//Roby - Alterado em 29/08/2020==========================INICIO==========================
// Entrada analógica 01 : NX6000_3 - %IW80 - Medição da temperatura da ENTRADA DA TORRE com SENSOR TIPO K e TXBLOCK =========================== 
converteEA103(IN:=EA103, IN_MIN:=0, IN_MAX:=4000,OUT_MIN:= -150, OUT_MAX:=1370);
TEMP_QUEIMATORRE:= converteEA103.OUT;

// Entrada analógica 02 : NX6000_3 - %IW82 - Medição da temperatura da SAÍDA ATMOSFERA com SENSOR TIPO K e TXBLOCK =========================== 
converteEA203(IN:=EA203, IN_MIN:=0, IN_MAX:=4000,OUT_MIN:= -150, OUT_MAX:=1370);
TEMP_QUEIMAATM:= converteEA203.OUT;

//Roby - Alterado em 23/02/2021==========================INÍCO==========================

// Entrada analógica 03 : NX6000_3 - %IW86 - Transdutor de pressão da tubulação óleo BPF. =========================== 
converteEA403(IN:=EA403, IN_MIN:=0, IN_MAX:=4000,OUT_MIN:=0, OUT_MAX:=16);
PRESS_OLEO_BPF:= converteEA403.OUT;
//Roby - Alterado em 23/02/2021==========================FIM==========================

// Entrada analógica 4 : NX6000_2 - Leitura Fluxo BBP02 ( dm³/h mA) ======================================================= 
converteEA502(IN:=EA502, IN_MIN:=0, IN_MAX:=4000,OUT_MIN:=0, OUT_MAX:=120);
VAZAO_VOLUMETRICA_REAL_BBP02:= converteEA502.OUT;

// Entrada analógica 4 : NX6000_2 - Leitura Fluxo BBP01 ( dm³/h mA) ======================================================= 
converteEA702(IN:=EA702, IN_MIN:=0, IN_MAX:=4000,OUT_MIN:=0, OUT_MAX:=120);
VAZAO_VOLUMETRICA_REAL_BBP01:= converteEA702.OUT;

END_PROGRAM

// Device/Application/BBP02
PROGRAM BBP02
VAR
	// Vazão volumetrica BBP02
	VAZAO_VOLUMETRICA_PRESET: REAL;
	// Vazão massica BBP02 kg/h
	VAZAO_MASSICA: REAL;
	//massa de dosagem do equipamento em Tonelada.
	MASSA:REAL;
	//Velocidade calculda do Dosador em Hz
	VELOCIDADE:REAL;
	//Espera o fluidizador baixar para o peso minino, pois atingiu o peso maximo
	ESPERA_FLUIDIZADOR_BAIXAR_PESO:BOOL;
	//Liga Dosador manual
	LIGA_DS_MANUAL:BOOL;
	//Liga Dosador automatico
	LIGA_DS_AUTO:BOOL;
	//Função de pulso do perfume
	PULSO_PERFUME:R_TRIG;
	// PID da BBP02
	PID_BBP02: NextoPID.PID;
	// constante
	A: BOOL;
	TMR_ATRASO_PERFUME: TON;
	INICIA_ATRASO_PERFUME: BOOL;
END_VAR

//   POU da bomba de perfume 2

//Controle manual ==========================================================

IF BTS_MAPH2 = FALSE THEN		
	
	//Bomba de perfume ===============================================
	//Formula
	//    Passo 1:     massa := (tonelada de dosagem * Percentual de dosagem(sem conversao)  * 10)  
	//    Passo 2:    Velocidade := ((massa + PRST_CONSTANTE_A_BBP02)/PRST_CONSTANTE_B_BBP02 
	//	  Inicialmente a Constante a:= -1.5
	//	  Inicialmente a Constante b:= 2.2948    	

	//calculo de velocidade  ======================================================
	IF MASSA_ESPECIFICA_BBP02 = 0 THEN
	MASSA_ESPECIFICA_BBP02 := 1;
	END_IF
	//Calcuulo da massa de dosagem do equipamento 
	MASSA := (PRST_VEL_PH2_MANUAL * 10 * PRST_PERC_DOSA_BBP02)/ MASSA_ESPECIFICA_BBP02;
	VAZAO_MASSICA := MASSA * MASSA_ESPECIFICA_BBP02;
	//Calculo da velocidade
	//VELOCIDADE := (MASSA + PRST_CONSTANTE_A_BBP02)/PRST_CONSTANTE_B_BBP02; 
	VELOCIDADE := MASSA; 
	IF BTS_BP2 = TRUE  AND AL_GERAL = FALSE   THEN
		IF LIGA_DS_MANUAL = TRUE THEN
			LIGA_DS_MANUAL := FALSE;
		ELSE
			LIGA_DS_MANUAL := TRUE;
		END_IF
		BTS_BP2 := FALSE;
	ELSIF AL_GERAL = TRUE THEN   //delsiga em caso de alarme
		LIGA_DS_MANUAL := FALSE;
		BTS_BP2 := FALSE;
	END_IF		
	
	//velocidde
	PRST_VEL_BPF2 := VELOCIDADE;
	VEL_PROGRAMADA_BBP02 := VAZAO_MASSICA;
	A := FALSE;
		
	//em manual desliga comando do automatico
	LIGA_DS_AUTO := FALSE;
ELSE	
	// controle automatico  =======================================================
		
	//Bomba de perfume ===============================================
	//Formula
	//    Passo 1:     massa := (tonelada de dosagem * Percentual de dosagem(sem conversao)  * 10)  
	//    Passo 2:    Velocidade := ((massa + PRST_CONSTANTE_A_BBP02)/PRST_CONSTANTE_B_BBP02 
	//	  Inicialmente a Constante a:= -1.5
	//	  Inicialmente a Constante b:= 2.2948    	

	//calculo de velocidade  ======================================================

	//Calcuulo da massa de dosagem do equipamento 
	MASSA := ((VELOCIDADE_PH2_AUTO/1000) * 10 * PRST_PERC_DOSA_BBP02)/ MASSA_ESPECIFICA_BBP02 ;
	VAZAO_MASSICA := MASSA;
	
	IF A = FALSE THEN	
		//Calculo da velocidade
		VELOCIDADE := (MASSA + PRST_CONSTANTE_A_BBP02)/PRST_CONSTANTE_B_BBP02; 
		A:=TRUE;
	END_IF	
	
	IF  AL_GERAL = FALSE   THEN		
		LIGA_DS_AUTO := TRUE;
	ELSE
		LIGA_DS_AUTO := FALSE;
	END_IF	
	
	//zera velocidade do ph com peso maximo
	IF LEITURA_PESO_FLUI2 >= PRST_PESO_MAX_FLUID2 THEN
		ESPERA_FLUIDIZADOR_BAIXAR_PESO := TRUE;
	END_IF
	
	//ativa velocidade do ph com peso minimo
	IF LEITURA_PESO_FLUI2 <= PRST_PESO_MIN_FLUID2 THEN
		ESPERA_FLUIDIZADOR_BAIXAR_PESO := FALSE;
	END_IF
	
	//se pode enviar peso 
//se pode enviar peso 
	IF ESPERA_FLUIDIZADOR_BAIXAR_PESO = FALSE THEN
		PRST_VEL_BPF2 := VELOCIDADE;
		VEL_PROGRAMADA_BBP02 := VAZAO_MASSICA;
		IF (VAZAO_VOLUMETRICA_REAL_BBP02 / MASSA_ESPECIFICA_BBP02) < (VAZAO_MASSICA - 1) THEN
			VELOCIDADE := VELOCIDADE + 0.1;
		END_IF
		IF (VAZAO_VOLUMETRICA_REAL_BBP02 / MASSA_ESPECIFICA_BBP02) > (VAZAO_MASSICA + 1) THEN
			VELOCIDADE := VELOCIDADE - 0.1;
		END_IF
		
	ELSE
		PRST_VEL_BPF2 := 0;
		VEL_PROGRAMADA_BBP02 := 0;
	END_IF
	
	//em auto desliga comando do manual
	LIGA_DS_MANUAL := FALSE;	
END_IF

//Liga dosador
IF LIGA_DS_AUTO = TRUE OR LIGA_DS_MANUAL = TRUE THEN
	INICIA_ATRASO_PERFUME := TRUE;
	VEL_BP2 := PRST_VEL_BPF2;
	LEITURA_VEL_BBP2 := VAZAO_VOLUMETRICA_REAL_BBP02/MASSA_ESPECIFICA_BBP02;
ELSE
	INICIA_ATRASO_PERFUME := FALSE;
	SD_BPER2 := FALSE;
	VEL_BP2:= 0;
	LEITURA_VEL_BBP2 := VAZAO_VOLUMETRICA_REAL_BBP02 / MASSA_ESPECIFICA_BBP02;
END_IF

//Atraso na partida da bomba de perfume para esperar chegada do pó.
TMR_ATRASO_PERFUME(IN:=INICIA_ATRASO_PERFUME,PT:= T#60S);
IF 	TMR_ATRASO_PERFUME.Q = TRUE AND LIGA_DS_AUTO = TRUE THEN
SD_BPER2 := TRUE;
END_IF

IF VEL_BP2 = 0 THEN 
	SD_BPER2 := FALSE;
END_IF
 
//Quantidade de consumo do perfume ===========================================

//gera pulso de contagem da agua		
PULSO_PERFUME(CLK:=ED_BP2);

//contador
IF PULSO_PERFUME.Q = TRUE THEN
	
	TOTALIZADOR1_BBP02 := TOTALIZADOR1_BBP02 + (PRST_RAZAO_BPF2 * MASSA_ESPECIFICA_BBP02 * 0.89);
	TOTALIZADOR2_BBP02 := TOTALIZADOR2_BBP02 + (PRST_RAZAO_BPF2 * MASSA_ESPECIFICA_BBP02 * 0.89);
	TOTALIZADOR3_BBP02 := TOTALIZADOR3_BBP02 + (PRST_RAZAO_BPF2 * MASSA_ESPECIFICA_BBP02 * 0.89);
	
END_IF

END_PROGRAM

// Device/Application/PH
PROGRAM PH
VAR
	//Tempos
	
	//Tempo de estrela do exaustor FM1
	TMR_ESTRELA_FM1:TON;
	//Tempo retardo troca de estrela para triangulo exaustor FM1
	TMR_RETARDO_TRIANGULO_FM1:TON;
	//Tempo de estrela do exaustor FM2
	TMR_ESTRELA_FM2:TON;
	//Tempo retardo troca de estrela para triangulo exaustor FM2
	TMR_RETARDO_TRIANGULO_FM2:TON;
	//Tempo de estrela do ventilador FM3
	TMR_ESTRELA_VFM2:TON;
	//Tempo retardo troca de estrela para triangulo ventilador FM2
	TMR_RETARDO_TRIANGULO_VFM2:TON;
	
	//Boleanos
	
	//Libera triangulo exaustor FM1
	LIBERA_TRIANGULO_FM1:BOOL;
	//Liga estrela exaustor FM1
	LIGA_ESTRELA_FM1:BOOL;
	//Liga triangulo exaustor FM1
	LIGA_TRIANGULO_FM1:BOOL;
	//Libera triangulo exaustor FM2
	LIBERA_TRIANGULO_FM2:BOOL;
	//Liga estrela exaustor FM2
	LIGA_ESTRELA_FM2:BOOL;
	//Liga triangulo exaustor FM2
	LIGA_TRIANGULO_FM2:BOOL;
	//Libera triangulo exaustor FM3
	LIBERA_TRIANGULO_VFM2:BOOL;
	//Liga estrela exaustor FM3
	LIGA_ESTRELA_VFM2:BOOL;
	//Liga triangulo exaustor FM3
	LIGA_TRIANGULO_VFM2:BOOL;
	//Liga exaustor FM1
	LIGA_FM1:BOOL;
	//Liga exaustor FM1
	LIGA_FM2:BOOL;
	//Liga ventilador FM2
	LIGA_VENTILADOR_FM2:BOOL;
	//Liga TC13
	LIGA_TC13:BOOL;
END_VAR

//     Processo Powder Handling - lógica do controle do PH

//=================================================================================================
// Controle manual dos equipamentos 
//=================================================================================================

//Controle manual PH 1

IF BTS_MAPH1 = FALSE THEN
	
	// Bomba de alimentação do oelo ===========================================	
	
	IF BTS_BALIOLEO = TRUE  AND AL_GERAL = FALSE  THEN	
		IF SD_BAO = TRUE THEN
			SD_BAO := FALSE;
		ELSE
			SD_BAO := TRUE;	
		END_IF
		 BTS_BALIOLEO := FALSE;
	END_IF
	//desliga em caso de alarme
	IF AL_GERAL = TRUE  THEN
		SD_BAO := FALSE;
		BTS_BALIOLEO := FALSE;
	END_IF
	
ELSE
	//=========================================================================
	// controle automatico PH1 
	//=========================================================================
	
	//Bomba alimentação do óleo ===============================================
	IF AL_GERAL = FALSE AND AL_GERAL = FALSE THEN
		SD_BAO := TRUE;
	ELSE
		SD_BAO := FALSE;
	END_IF
		
END_IF


//=================================================================================================
// Controles que independem do manual/automatico 
//=================================================================================================


// Ventilador do Fluidizador ================================================
//Velocidade  de 0-100%

IF BTS_VENTIFLUIDIZADOR = TRUE  AND AL_GERAL=FALSE THEN
	IF SD_VFLU = TRUE THEN
		SD_VFLU := FALSE;
	ELSE
		SD_VFLU := TRUE;
	END_IF	
	BTS_VENTIFLUIDIZADOR := FALSE;
END_IF
//delsiga em caso de alarme
IF AL_GERAL = TRUE THEN
	SD_VFLU := FALSE;
END_IF

//move velocidade
IF SD_VFLU = TRUE THEN
	VEL_VENTFLUIDIZADOR := PRST_VEL_VENTIFLUIDIZADOR;
ELSE
	VEL_VENTFLUIDIZADOR := 0;
END_IF


//Exaustor FM1 ========================================================

IF BTS_EXFM1 = TRUE AND AL_EXFM1_E = FALSE AND AL_GERAL = FALSE THEN
		IF LIGA_FM1 = TRUE THEN
			LIGA_FM1 := FALSE;
		ELSE
			LIGA_FM1 := TRUE;
		END_IF		
		BTS_EXFM1 := FALSE;	
ELSIF AL_GERAL = TRUE THEN
	LIGA_FM1 := FALSE;
	BTS_EXFM1 := FALSE;
END_IF

//comando estrela/triangulo
//LIGA ESTRELA	
IF LIGA_FM1 = TRUE AND AL_EXFM1_E = FALSE AND  AL_GERAL = FALSE THEN
	IF LIGA_ESTRELA_FM1 = FALSE THEN
		//Contatora estrela
		SD_EXFM1_E := TRUE;
	ELSE
		//Contatora estrela
		SD_EXFM1_E := FALSE;
	END_IF
	LIBERA_TRIANGULO_FM1 := TRUE;
ELSE
	//Contatora estrela
	SD_EXFM1_E := FALSE;	
	LIBERA_TRIANGULO_FM1:=FALSE;
END_IF
	
//TEMPO PARA ENTRAR O TRIANGULO
TMR_ESTRELA_FM1(IN:= LIBERA_TRIANGULO_FM1, PT:= T#6S);	
LIGA_ESTRELA_FM1 := TMR_ESTRELA_FM1.Q;
//TEMPO DE INTERVALO ENTRE ESTRELA E TRIANGULO
TMR_RETARDO_TRIANGULO_FM1(IN:= LIGA_ESTRELA_FM1, PT:= T#0.2S);
LIGA_TRIANGULO_FM1 := TMR_RETARDO_TRIANGULO_FM1.Q;
//Contatora triangulo
SD_EXFM1_T := LIGA_TRIANGULO_FM1;

//contatora Principal	
IF LIBERA_TRIANGULO_FM1 = TRUE THEN
	SD_EXFM1_P := TRUE;
ELSE
	SD_EXFM1_P := FALSE;
END_IF

//Exaustor FM2 ========================================================

IF BTS_EXFM2 = TRUE AND AL_EXFM1_E = FALSE AND AL_GERAL = FALSE THEN
		IF LIGA_FM2 = TRUE THEN
			LIGA_FM2 := FALSE;
		ELSE
			LIGA_FM2 := TRUE;
		END_IF		
		BTS_EXFM2 := FALSE;	
ELSIF AL_GERAL = TRUE THEN
	LIGA_FM2 := FALSE;
	BTS_EXFM2 := FALSE;	
END_IF

//comando estrela/triangulo
//LIGA ESTRELA	
IF LIGA_FM2 = TRUE AND AL_EXFM2_E = FALSE  AND AL_EXFM2_T = FALSE AND AL_GERAL = FALSE THEN
	IF LIGA_ESTRELA_FM2 = FALSE THEN
		//Contatora estrela
		SD_EXFM2_E := TRUE;
	ELSE
		//Contatora estrela
		SD_EXFM2_E := FALSE;
	END_IF
	LIBERA_TRIANGULO_FM2 := TRUE;
ELSE
	//Contatora estrela
	SD_EXFM2_E := FALSE;	
	LIBERA_TRIANGULO_FM2:=FALSE;
END_IF
	
//TEMPO PARA ENTRAR O TRIANGULO
TMR_ESTRELA_FM2(IN:= LIBERA_TRIANGULO_FM2, PT:= T#6S);	
LIGA_ESTRELA_FM2 := TMR_ESTRELA_FM2.Q;
//TEMPO DE INTERVALO ENTRE ESTRELA E TRIANGULO
TMR_RETARDO_TRIANGULO_FM2(IN:= LIGA_ESTRELA_FM2, PT:= T#0.2S);
LIGA_TRIANGULO_FM2 := TMR_RETARDO_TRIANGULO_FM2.Q;
//Contatora triangulo
SD_EXFM2_T := LIGA_TRIANGULO_FM2;

//contatora Principal	
IF LIBERA_TRIANGULO_FM2 = TRUE THEN
	SD_EXFM2_P := TRUE;
ELSE
	SD_EXFM2_P := FALSE;
END_IF


//Ventilador FM1 - PH1 ========================================================

IF BTS_EXVFM2 = TRUE AND AL_EXFM1_E = FALSE AND  AL_GERAL = FALSE THEN
		IF LIGA_VENTILADOR_FM2 = TRUE THEN
			LIGA_VENTILADOR_FM2 := FALSE;
		ELSE
			LIGA_VENTILADOR_FM2 := TRUE;
		END_IF		
		BTS_EXVFM2 := FALSE;
ELSIF  AL_GERAL = TRUE THEN
	LIGA_VENTILADOR_FM2 := FALSE;
	BTS_EXVFM2 := FALSE;
END_IF


//comando estrela/triangulo
//LIGA ESTRELA	
IF LIGA_VENTILADOR_FM2 = TRUE AND AL_VEXFM2_E = FALSE AND AL_VEXFM2_T = FALSE AND  AL_GERAL = FALSE THEN
	IF LIGA_ESTRELA_VFM2 = FALSE THEN
		//Contatora estrela
		SD_VEXFM2_E := TRUE;
	ELSE
		//Contatora estrela
		SD_VEXFM2_E := FALSE;
	END_IF
	LIBERA_TRIANGULO_VFM2 := TRUE;
ELSE
	//Contatora estrela
	SD_VEXFM2_E := FALSE;	
	LIBERA_TRIANGULO_VFM2:=FALSE;
END_IF
	
//TEMPO PARA ENTRAR O TRIANGULO
TMR_ESTRELA_VFM2(IN:= LIBERA_TRIANGULO_VFM2, PT:= T#6S);	
LIGA_ESTRELA_VFM2 := TMR_ESTRELA_VFM2.Q;
//TEMPO DE INTERVALO ENTRE ESTRELA E TRIANGULO
TMR_RETARDO_TRIANGULO_VFM2(IN:= LIGA_ESTRELA_VFM2, PT:= T#0.2S);
LIGA_TRIANGULO_VFM2 := TMR_RETARDO_TRIANGULO_VFM2.Q;
//Contatora triangulo
SD_VEXFM2_T := LIGA_TRIANGULO_VFM2;

//contatora Principal	
IF LIBERA_TRIANGULO_VFM2 = TRUE THEN
	SD_VEXFM2_P := TRUE;
ELSE
	SD_VEXFM2_P := FALSE;
END_IF

//Ventilador FM2 - PH2 ========================================================

IF BTS_VENTIFLUIDIZADOR = TRUE AND AL_GERAL = FALSE THEN
	IF SD_VFLU = TRUE THEN
		SD_VFLU := FALSE;
	ELSE
		SD_VFLU := TRUE;
	END_IF		
	BTS_VENTIFLUIDIZADOR := FALSE;	
ELSIF AL_GERAL = TRUE THEN
	SD_VFLU := FALSE;
	BTS_VENTIFLUIDIZADOR := FALSE;
END_IF

//Esteira TC8 ===============================================================

IF BTS_ESTTC8 = TRUE  AND AL_GERAL = FALSE AND SD_ESTTC8_R = FALSE  THEN	
	IF SD_ESTTC8 = TRUE THEN
		SD_ESTTC8 := FALSE;	
	ELSE
		SD_ESTTC8 := TRUE;
	END_IF	
	BTS_ESTTC8 := FALSE;
END_IF
//desliga em caso de alarme
IF AL_GERAL = TRUE  THEN
	SD_ESTTC8 := FALSE;	
	BTS_ESTTC8 := FALSE;
END_IF

//Reversão
IF BTS_ESTTC8REVER = TRUE  AND AL_GERAL=FALSE AND SD_ESTTC8 = FALSE THEN	
	IF SD_ESTTC8_R = TRUE THEN
		SD_ESTTC8_R := FALSE;
	ELSE
		SD_ESTTC8_R := TRUE;
	END_IF
		BTS_ESTTC8REVER := FALSE;
END_IF
//desliga em caso de alarme
IF AL_GERAL = TRUE THEN
	SD_ESTTC8_R := FALSE;	
	BTS_ESTTC8REVER := FALSE;
END_IF


//Esteira po base 1 ========================================================
IF LIGA_DS1 = TRUE AND AL_GERAL=FALSE THEN
	SD_ESTPOB1 := TRUE;
ELSE
	SD_ESTPOB1 := FALSE;
END_IF


//Esteria Po base 11 =========================================================

IF LIGA_DS11 = TRUE AND AL_GERAL = FALSE  THEN
	SD_ESTPOB11 := TRUE;
ELSE
	SD_ESTPOB11 := FALSE;
END_IF


//Esteira TC9 ================================================================

IF (SD_DS6 = TRUE OR LIGA_DS4= TRUE OR LIGA_DS5 = TRUE) AND AL_GERAL = FALSE THEN
	SD_ESTTC9 := TRUE;
ELSE
	SD_ESTTC9 := FALSE;
END_IF


//Esteira TC10 ================================================================

IF (LIGA_DS2= TRUE OR LIGA_DS3 = TRUE) AND AL_GERAL = FALSE THEN
	SD_ESTTC10 := TRUE;
ELSE
	SD_ESTTC10 := FALSE;
END_IF


//Esteira TC12 ================================================================

IF (LIGA_DS10 = TRUE OR LIGA_DS12 = TRUE OR LIGA_DS14) AND AL_GERAL = FALSE THEN
	SD_ESTTC12 := TRUE;
ELSE
	SD_ESTTC12 := FALSE;
END_IF

//Esteira TC13 ==============================================================
			
	IF (LIGA_TC13 = TRUE OR LIGA_DS8 = TRUE OR LIGA_DS9 = TRUE) AND AL_GERAL = FALSE THEN
 		SD_ESTTC13 := TRUE;
	ELSE
		SD_ESTTC13 := FALSE;
	END_IF

//Elevador 2 ================================================================

IF BTS_EL2 = TRUE AND AL_GERAL = FALSE  THEN
	IF SD_EL2DMIX= TRUE THEN		
		SD_EL2DMIX := false;
	ELSE		
		SD_EL2DMIX :=TRUE;
	END_IF
	BTS_EL2 := FALSE;	
END_IF 
//desliga em caso de alarme
IF AL_GERAL = TRUE  THEN
	SD_EL2DMIX:= FALSE;
	BTS_EL2 := FALSE;
END_IF

//Elevador 4 ==================================================================

IF BTS_EL4 = TRUE AND AL_GERAL = FALSE  THEN
	IF SD_EL2= TRUE THEN
		SD_EL2:= FALSE;		
	ELSE
		SD_EL2:= TRUE;		
	END_IF
	BTS_EL4 := FALSE;	
END_IF 
//desliga em caso de alarme
IF AL_GERAL = TRUE  THEN
	SD_EL2:= FALSE;
	BTS_EL4 := FALSE;	
END_IF


//Peneiras ====================================================================

//1
IF BTS_PNS AND AL_GERAL = FALSE THEN
	IF SD_M1PN= TRUE THEN
		SD_M1PN:= FALSE;
	ELSE
		SD_M1PN:= TRUE;
	END_IF
	BTS_PNS :=FALSE;	
END_IF
//desliga em caso de alarme
IF AL_GERAL = TRUE THEN
	SD_M1PN := FALSE;	
END_IF

IF SD_M1PN = TRUE THEN
	SD_M2PN:= TRUE;
	SD_M3PN:= TRUE;
	SD_M4PN:= TRUE;
ELSE
	SD_M2PN:= FALSE;
	SD_M3PN:= FALSE;
	SD_M4PN:= FALSE;
END_IF


//Esteira TC13 ================================================================

IF BTS_ESTTC13 = TRUE AND SD_EL2DMIX = TRUE AND AL_GERAL = FALSE THEN
	IF SD_ESTTC13 = TRUE THEN
		SD_ESTTC13 := FALSE;
	ELSE
		SD_ESTTC13 := TRUE;	
	END_IF
	BTS_ESTTC13 := FALSE;
ELSIF  AL_GERAL = TRUE THEN
	SD_ESTTC13 := FALSE;
	BTS_ESTTC13 := FALSE;
END_IF


//Esteira TC3 Dry Mix =========================================================

IF BTS_TC3 = TRUE AND SD_EL2DMIX = TRUE AND AL_GERAL = FALSE THEN
	IF SD_ESTTC3 = TRUE THEN
		SD_ESTTC3 := FALSE;
	ELSE
		SD_ESTTC3 := TRUE;	
	END_IF
	BTS_TC3 := FALSE;
ELSIF SD_EL2DMIX = FALSE THEN
	SD_ESTTC3 := FALSE;
	BTS_TC3 := FALSE;
END_IF
//desliga em caso de alarme
IF AL_GERAL = TRUE  THEN
	SD_ESTTC3:= FALSE;
	BTS_TC3 := FALSE;
END_IF

//=============================================================================
// Fluidizadores
//=============================================================================
//habilita / Desabilita Fluidizador conforme peso

//Fluidizador 1 ===============================================================

//Desabilita fluidizador 
IF LEITURA_PESO_FLUI1 > PRST_PESO_MAX_FLUID1  THEN		
	DESLIGA_FLUIDIZADOR1 := TRUE;
END_IF
//Habilita fluidizador 1
IF LEITURA_PESO_FLUI1 < PRST_PESO_MIN_FLUID1 THEN
	DESLIGA_FLUIDIZADOR1 := FALSE;
END_IF


//Fluidizador 2 ==============================================================

//Desabilita fluidizador 
IF LEITURA_PESO_FLUI2 >= PRST_PESO_MAX_FLUID2  THEN		
	DESLIGA_FLUIDIZADOR2 := TRUE;
END_IF
//Habilita fluidizador 
IF LEITURA_PESO_FLUI2 <= PRST_PESO_MIN_FLUID2 THEN
	DESLIGA_FLUIDIZADOR2 := FALSE;
END_IF

END_PROGRAM

// Device/Application/BBP01
PROGRAM BBP01
VAR
	Teste: REAL;
	VAZAO_VOLUMETRICA_PRESET: REAL;
	//massa de dosagem do equipamento em Tonelada.
	MASSA:REAL;
	//Velocidade calculda do Dosador em Hz
	VELOCIDADE:REAL;
	//Espera o fluidizador baixar para o peso minino, pois atingiu o peso maximo
	ESPERA_FLUIDIZADOR_BAIXAR_PESO:BOOL;
	//Liga Dosador manual
	LIGA_DS_MANUAL:BOOL;
	//Liga Dosador automatico
	LIGA_DS_AUTO:BOOL;
	//Função de pulso do perfume
	PULSO_PERFUME:R_TRIG;
	// Vazão massica da bomba de perfume 1 (kg/h)
	VAZAO_MASSICA: REAL;
	// PID da Bomba de perfume 1
	PID_BBP01: NextoPID.PID;
	// VARIÁVEL AUXILIAR
	A: BOOL;
	b: REAL;
	TMR_ATRASO_PERFUME: TON;
	INICIA_ATRASO_PERFUME: BOOL;
END_VAR

//   POU da bomba de perfme 1

//Controle manual ==========================================================

IF BTS_MAPH1 = FALSE THEN	
	
	//Bomba de perfume - sistema antigo ===============================================
	//Formula
	//    Passo 1:     massa := (tonelada de dosagem * Percentual de dosagem(sem conversao)  * 10)  
	//    Passo 2:    Velocidade := ((massa + PRST_CONSTANTE_A_BBP01)/PRST_CONSTANTE_B_BBP01 
	//	  Inicialmente a Constante a:= -1.5
	//	  Inicialmente a Constante b:= 2.2948      	

	//calculo de velocidade  ======================================================

	//Calcuulo da massa de dosagem do equipamento 
		IF MASSA_ESPECIFICA_BBP01 = 0 THEN
		MASSA_ESPECIFICA_BBP01 := 1;
		END_IF
	MASSA := (PRST_VEL_PH1_MANUAL * 10 * PRST_PERC_DOSA_BBP01) / MASSA_ESPECIFICA_BBP01;
	
	//Vazão volumetrica calculada
	VAZAO_MASSICA := MASSA * MASSA_ESPECIFICA_BBP01;
	
	//Calculo da velocidade
	//VELOCIDADE := (MASSA + PRST_CONSTANTE_A_BBP01)/PRST_CONSTANTE_B_BBP01; 
		VELOCIDADE := MASSA ; 
	//Manual
	IF BTS_BP1 = TRUE  AND AL_GERAL = FALSE   THEN
		IF LIGA_DS_MANUAL = TRUE THEN
			LIGA_DS_MANUAL := FALSE;
		ELSE
			LIGA_DS_MANUAL := TRUE;
		END_IF
		BTS_BP1 := FALSE;
	ELSIF AL_GERAL = TRUE THEN  //delsiga em caso de alarme
		LIGA_DS_MANUAL := FALSE;
		BTS_BP1 := FALSE;
	END_IF
	
	//velocidde
	PRST_VEL_BPF1 := VELOCIDADE;
	VEL_PROGRAMADA_BBP01 := VAZAO_MASSICA ;
	A := FALSE;
	
	//em manual desliga comando do automatico
	LIGA_DS_AUTO := FALSE;
ELSE	
	// controle automatico PH1 =================================================	
	
	//Bomba de perfume - sistema antigo ===============================================
	//Formula
	//    Passo 1:     massa := (tonelada de dosagem * Percentual de dosagem(sem conversao)  * 10)  
	//    Passo 2:    Velocidade := ((massa + PRST_CONSTANTE_A_BBP01)/PRST_CONSTANTE_B_BBP01 
	//	  Inicialmente a Constante a:= -1.5
	//	  Inicialmente a Constante b:= 2.2948      	

	//calculo de velocidade  ======================================================
	//Calcuulo da massa de dosagem do equipamento 
	MASSA := ((VELOCIDADE_PH1_AUTO / 1000) * 10 * PRST_PERC_DOSA_BBP01) / MASSA_ESPECIFICA_BBP01;
	VAZAO_MASSICA := MASSA;
	IF A = FALSE THEN	
		//Calculo da velocidade
		VELOCIDADE := (MASSA + PRST_CONSTANTE_A_BBP01)/PRST_CONSTANTE_B_BBP01; 
		A:=TRUE;
	END_IF	
		
	IF  AL_GERAL = FALSE   THEN
		LIGA_DS_AUTO := TRUE;
	ELSE
		LIGA_DS_AUTO := FALSE;
	END_IF	
	
	//zera velocidade do ph com peso maximo
	IF LEITURA_PESO_FLUI1 >= PRST_PESO_MAX_FLUID1 THEN
		ESPERA_FLUIDIZADOR_BAIXAR_PESO := TRUE;
	END_IF
	
	//ativa velocidade do ph com peso minimo
	IF LEITURA_PESO_FLUI1 <= PRST_PESO_MIN_FLUID1 THEN
		ESPERA_FLUIDIZADOR_BAIXAR_PESO := FALSE;
	END_IF
	
	//se pode enviar peso 
	IF ESPERA_FLUIDIZADOR_BAIXAR_PESO = FALSE THEN
		PRST_VEL_BPF1 := VELOCIDADE;
		VEL_PROGRAMADA_BBP01 := VAZAO_MASSICA;
		IF (VAZAO_VOLUMETRICA_REAL_BBP01/MASSA_ESPECIFICA_BBP01) < (VAZAO_MASSICA - 1) THEN
			VELOCIDADE := VELOCIDADE + 0.1;
		END_IF
		IF (VAZAO_VOLUMETRICA_REAL_BBP01/MASSA_ESPECIFICA_BBP01) > (VAZAO_MASSICA + 1) THEN
			VELOCIDADE := VELOCIDADE - 0.1;
		END_IF
		
	ELSE
		PRST_VEL_BPF1 := 0;
		VEL_PROGRAMADA_BBP01 := 0;
	END_IF
	
	//em auto desliga comando do manual
	LIGA_DS_MANUAL := FALSE;
END_IF

//Liga dosador
IF LIGA_DS_AUTO = TRUE OR LIGA_DS_MANUAL = TRUE THEN
	INICIA_ATRASO_PERFUME := TRUE;
	VEL_BP1 := PRST_VEL_BPF1;
	LEITURA_VEL_BBP1 := VAZAO_VOLUMETRICA_REAL_BBP01/MASSA_ESPECIFICA_BBP01;

ELSE
	INICIA_ATRASO_PERFUME := FALSE;
	SD_BPER1 := FALSE;
	VEL_BP1:= 0;
	LEITURA_VEL_BBP1 := VAZAO_VOLUMETRICA_REAL_BBP01/MASSA_ESPECIFICA_BBP01;
END_IF
	//Atraso na partida da bomba de perfume para esperar chegada do pó.
TMR_ATRASO_PERFUME(IN:=INICIA_ATRASO_PERFUME,PT:= T#40S);
IF 	TMR_ATRASO_PERFUME.Q = TRUE AND LIGA_DS_AUTO = TRUE THEN
SD_BPER1 := TRUE;
END_IF

IF VEL_BP1 = 0 THEN 
	SD_BPER1 := FALSE;
END_IF
//Quantidade de consumo do perfume ===========================================

//gera pulso de contagem da agua		
PULSO_PERFUME(CLK:=ED_BP1);

//contador
IF PULSO_PERFUME.Q = TRUE THEN
	
	TOTALIZADOR1_BBP01 := TOTALIZADOR1_BBP01 + (PRST_RAZAO_BPF1 * MASSA_ESPECIFICA_BBP01 * 0.73);
	TOTALIZADOR2_BBP01 := TOTALIZADOR2_BBP01 + (PRST_RAZAO_BPF1 * MASSA_ESPECIFICA_BBP01 * 0.73);
	TOTALIZADOR3_BBP01 := TOTALIZADOR3_BBP01 + (PRST_RAZAO_BPF1 * MASSA_ESPECIFICA_BBP01 * 0.73);
	
END_IF

END_PROGRAM

// Device/Application/Temperturas
PROGRAM Temperturas

//Move as temperaturas das entrads analogicas para região temporaria dividindo por 10 para gerar o ponto.

//Temperatura do vapor
TEMP_VAPOR := (TEMPVAPOR / 10)-9;
//Temperatura da torre
//TEMP_TORRE := TEMPTORE / 10;
//TEMPERATURA_TORRE := TEMPTORE / 10;;
//Temperatura do queimador para torre
//TEMP_QUEIMATORRE := ((TEMPQUEIMATORRE / 10) * 1.197);
//Temperatura do queimador para atmosfera
//TEMP_QUEIMAATM := TEMPQUEIMADORATM / 10;

END_PROGRAM

// Device/Application/SlurryMaking
PROGRAM SlurryMaking
VAR
	//Temporizadores

	//Tempo de estrela do mexedor principal
	TMR_ESTRELA_MXP:TON;
	//Tempo retardo troca de estrela para triangulo mexedor principal
	TMR_RETARDO_TRIANGULO_MXP:TON;		
	//Tempo de reação
	TMR_REACAO:TON;
	//Tempo de hidratação
	TMR_HIDRATA:TON;
	//Tempo de homogenizacao
	TMR_HOMOGE:TON;
	//Tempo retardo troca de sequencia
	TMR_TROCA_SEQUENCIA:TON;
	
	//Tempo reação em TIME
	TEMPO_REACAO:TIME;
	//Tempo reação em REAL temporario para multiplicar por 1000
	TEMPO_REACAO_TEMPORARIO:REAL;
	//Tempo de hidratação em TIME
	TEMPO_HIDRATA:TIME;
	//Tempo de hidratação em REAL Temporario para multiplicar por 1000
	TEMPO_HIDRATA_TEMPORARIO:REAL;
	//Tempo de Homogenização em TIME
	TEMPO_HOMOGE:TIME;
	//Tempo de Homogenização em REAL temporario para multiplicar por 1000
	TEMPO_HOMOGE_TEMPORARIO:REAL;
	//Peso do Blend com Acusol
	PESO_BLL4_ACUSOL:REAL;
	
	
	//Boleanos
	
	//Liga Mexedor
	LIGA_MEXEDOR:BOOL;
	//Libera triangulo mexedor principal
	LIBERA_TRIANGULO_MXP:BOOL;
	//Liga estrela mexedor principal
	LIGA_ESTRELA_MXP:BOOL;
	//Liga triangulo mexedor principal
	LIGA_TRIANGULO_MXP:BOOL;
	//Informa que ja contou a agua
	JA_CONTOU_AGUA:BOOL;
	//Ciclo em processo
	CICLO_PROCESSO:BOOL;
	//Iniciar tempo de reação
	INICIAR_TEMPO_REACAO:BOOL;
	//Iniciar tempo de hidratacao
	INICIAR_TEMPO_HIDRATACAO:BOOL;
	//Iniciar tempo de homogenizacao
	INICIAR_TEMPO_HOMOGENIZACAO:BOOL;
	//Libera tempo de intervalo de troca de sequencia
	INTERVALO_TROCA_SEQUE:BOOL;
	//Habilita continuidade da sequencia
	CONTINUA_SEQUENCIA:BOOL;
	//Liga controle de temperatura no mexedor principal
	LIGA_CONTROLE_TEMPERATURA_MXP:BOOL;
	//Ultima batelada
	ULTIMA_BATELADA:BOOL;
	//libera carregar as balanças antes do ciclo iniciar
	CARREGA_BALANCA_ANTESINICIOCICLO:BOOL;
	//Fim de produção
	FIM_PRODUCAO:BOOL;	
	//Agua dosada
	AGUA_DOSADA:BOOL;
	//reset contador agua em automatico
	RESET_AGUA_AUTO:BOOL;
	//reset contador agua
	RESET_AGUA:BOOL;
	//descarga iniciada BLS1
	DESCARGA_INICIADA_BLS1:BOOL;
	//descarga iniciada BLS2
	DESCARGA_INICIADA_BLS2:BOOL;
	//descarga iniciada BLS3
	DESCARGA_INICIADA_BLS3:BOOL;
	//descarga iniciada BLS4
	DESCARGA_INICIADA_BLS4:BOOL;
	//descarga iniciada BLS5
	DESCARGA_INICIADA_BLS5:BOOL;
	//descarga iniciada BLL1
	DESCARGA_INICIADA_BLL1:BOOL;
	//descarga iniciada BLL2
	DESCARGA_INICIADA_BLL2:BOOL;
	//descarga iniciada BLL3
	DESCARGA_INICIADA_BLL3:BOOL;
	//descarga iniciada BLL4
	DESCARGA_INICIADA_BLL4:BOOL;
	//Leitura de produção realizada BLS1
	LEITURA_REALIZADA_BLS1:BOOL;
	//Leitura de produção realizada BLS2
	LEITURA_REALIZADA_BLS2:BOOL;
	//Leitura de produção realizada BLS3
	LEITURA_REALIZADA_BLS3:BOOL;
	//Leitura de produção realizada BLS4
	LEITURA_REALIZADA_BLS4:BOOL;
	//Leitura de produção realizada BLS5
	LEITURA_REALIZADA_BLS5:BOOL;
	//Leitura de produção realizada BLL1
	LEITURA_REALIZADA_BLL1:BOOL;
	//Leitura de produção realizada BLL2
	LEITURA_REALIZADA_BLL2:BOOL;
	//Leitura de produção realizada BLL3
	LEITURA_REALIZADA_BLL3:BOOL;
	//Leitura de produção realizada BLL4
	LEITURA_REALIZADA_BLL4:BOOL;
	//Leitura de produção realizada Agua
	LEITURA_REALIZADA_AGUA:BOOL;
	
	//Funções de Triger

	//Função de pulso da agua
	PULSO_AGUA:R_TRIG;
	//Pulso inicio de ciclo
	PULSO_INICIO_CICLO:R_TRIG;
	//Pulso Balança de solido 1 carregada
	PULSO_BLS1_CARREGADA:R_TRIG;
	//Pulso Balança de solido 2 carregada
	PULSO_BLS2_CARREGADA:R_TRIG;
	//Pulso Balança de solido 3 carregada
	PULSO_BLS3_CARREGADA:R_TRIG;
	//Pulso Balança de solido 4 carregada
	PULSO_BLS4_CARREGADA:R_TRIG;
	//Pulso Balança de solido 5 carregada
	PULSO_BLS5_CARREGADA:R_TRIG;
	//Pulso Balança de liquido 1 carregada
	PULSO_BLL1_CARREGADA:R_TRIG;
	//Pulso Balança de liquido 2 carregada
	PULSO_BLL2_CARREGADA:R_TRIG;
	//Pulso Balança de liquido 3 carregada
	PULSO_BLL3_CARREGADA:R_TRIG;
	//Pulso Balança de liquido 4 carregada
	PULSO_BLL4_CARREGADA:R_TRIG;
	

	//Contadores
	
	//Contador de pulsos de agua
	CONTADOR_AGUA:TON;
	
	
	
	//Contagem real de pulsos do contador
	CV:INT;	
	// Temporizador
	QNTDADE_PULSOS_AGUA:TIME;
	// Conversão de tempo para litros
	QNTDADE_PULSOS_AGUA_REAL: REAL;
	// Temporizador em tempo real
	ET: TIME;
	// Resultado mostrado no supervisório da quantidade em litros dosada em tempo real
	TMR_AGUA_DOSADA: REAL;
	//PARADA DA ESTEIRA INCLINADA 
	TM_SD_R7: TON;
	TM_AUX_SD_R7: TIME;
	SD_R7_AUX: BOOL;
END_VAR

//     Processo Slurry Making - lógica do controle da preparação de pasta

//================================ Controle manual dos equipamentos ===========================================================================

IF AL_GERAL = TRUE THEN
	BTS_MASLU := FALSE;
END_IF

//apresenta a posicao real da sequencia do slurry =================================
LEITURA_SEQ_ATUAL := INT_TO_REAL(CNT_SEQUENCIA_SLURRY);


IF BTS_MASLU = FALSE THEN

	//Carregamento das balanças  

	//Rosca de po 1 ============================================================
	IF BTS_RPO1 = TRUE  AND AL_GERAL = FALSE AND SD_BLS1 = FALSE THEN
		IF SD_RPO1 = TRUE THEN
			SD_RPO1 := FALSE;	
		ELSE
			SD_RPO1 := TRUE;			
		END_IF		
		BTS_RPO1 := FALSE;	
	ELSIF AL_GERAL = TRUE AND SD_BLS1 = TRUE THEN      //desliga se alarmes
		SD_RPO1 := FALSE;
		BTS_RPO1 := FALSE;
	END_IF
	//Desliga a rosca automaticamente pelo peso
	IF SD_RPO1 = TRUE AND LEITURA_PESO_BLS1 > PRST_PESO_BLS1 THEN
		SD_RPO1 := FALSE;
	END_IF
	

	//Rosca de po 2 ================================================================
	IF BTS_RPO2 = TRUE AND AL_GERAL = FALSE AND SD_BLS2 = FALSE THEN
		IF SD_RPO2 = TRUE THEN
			SD_RPO2 := FALSE;	
		ELSE
			SD_RPO2 := TRUE;
		END_IF		
		BTS_RPO2 := FALSE;	
	ELSIF AL_GERAL = TRUE AND SD_BLS1 = TRUE THEN      //desliga se alarmes
		SD_RPO1 := FALSE;	
		BTS_RPO2 := FALSE;
	END_IF
	//Desliga a rosca automaticamente pelo peso
	IF SD_RPO2 = TRUE AND LEITURA_PESO_BLS2 > PRST_PESO_BLS2 THEN
		SD_RPO2 := FALSE;
	END_IF

	//Rosca de po 3 =================================================================
	IF BTS_RPO3 = TRUE  AND AL_GERAL = FALSE AND SD_BLS3 = FALSE THEN
		IF SD_RPO3 = TRUE THEN
			SD_RPO3 := FALSE;	
		ELSE
			SD_RPO3 := TRUE;
		END_IF		
		BTS_RPO3 := FALSE;
	ELSIF  AL_GERAL = TRUE AND SD_BLS1 = TRUE THEN //desliga se alarmes
		SD_RPO3 := FALSE;
		BTS_RPO3 := FALSE;
	END_IF
	//Desliga a rosca automaticamente pelo peso
	IF SD_RPO3 = TRUE AND LEITURA_PESO_BLS3 > PRST_PESO_BLS3 THEN
		SD_RPO3 := FALSE;
	END_IF

	//Rosca de po 4 =================================================================
	IF BTS_RPO4 = TRUE  AND AL_GERAL = FALSE AND SD_BLS4 = FALSE THEN
		IF SD_RPO4 = TRUE THEN
			SD_RPO4 := FALSE;	
		ELSE
			SD_RPO4 := TRUE;
		END_IF		
		BTS_RPO4 := FALSE;	
	ELSIF AL_GERAL = TRUE AND SD_BLS1 = TRUE THEN //desliga se alarmes
		SD_RPO4 := FALSE;
		BTS_RPO4 := FALSE;		
	END_IF
	//Desliga a rosca automaticamente pelo peso
	IF SD_RPO4 = TRUE AND LEITURA_PESO_BLS4 > PRST_PESO_BLS4 THEN
		SD_RPO4 := FALSE;
	END_IF

	//Rosca de po 5 =================================================================
	IF BTS_RPO5 = TRUE  AND AL_GERAL = FALSE AND SD_BLS5 = FALSE THEN
		IF SD_RPO5 = TRUE THEN
			SD_RPO5 := FALSE;	
		ELSE
			SD_RPO5 := TRUE;
		END_IF		
		BTS_RPO5 := FALSE;	
	ELSIF  AL_GERAL = TRUE AND SD_BLS5 = TRUE THEN //desliga se alarmes
		SD_RPO5 := FALSE;	
		BTS_RPO5 := FALSE;
	END_IF
	//Desliga a rosca automaticamente pelo peso
	IF SD_RPO5 = TRUE AND LEITURA_PESO_BLS5 > PRST_PESO_BLS5 THEN
		SD_RPO5 := FALSE;
	END_IF

	//Balança liquidos 1 - carga rapida  ============================================
	IF BTS_BLL1R = TRUE  AND SD_BLL1D = FALSE AND AL_GERAL = FALSE THEN
		IF SD_BLL1R = TRUE THEN
			SD_BLL1R := FALSE;
		ELSE
			SD_BLL1R := TRUE;	
		END_IF		
		BTS_BLL1R := FALSE;	
	ELSIF  AL_GERAL = TRUE THEN //desliga se alarmes
		SD_BLL1R := FALSE;
		BTS_BLL1R := FALSE;	
	END_IF

	//Balança liquidos 1 - carga lenta
	IF BTS_BLL1L = TRUE AND  SD_BLL1D = FALSE AND AL_GERAL = FALSE THEN
		IF SD_BLL1L = TRUE THEN
			SD_BLL1L := FALSE;
		ELSE
			SD_BLL1L := TRUE;
		END_IF		
		BTS_BLL1L := FALSE;	
	ELSIF  AL_GERAL = TRUE THEN //desliga se alarmes
		SD_BLL1L := FALSE;
		BTS_BLL1L := FALSE;
	END_IF
	
	//Desliga a rosca automaticamente pelo peso
	IF (SD_BLL1L = TRUE OR SD_BLL1R = TRUE) AND LEITURA_PESO_BLL1 > PRST_PESO_BLL1 THEN
		SD_BLL1L := FALSE;
		SD_BLL1R := FALSE;
	END_IF


	//Balança liquidos 2 - carga rapida ============================================
	IF BTS_BLL2R = TRUE  AND SD_BLL2D = FALSE AND AL_GERAL = FALSE THEN
		IF SD_BLL2R = TRUE THEN
			SD_BLL2R := FALSE;
		ELSE
			SD_BLL2R := TRUE;
		END_IF		
		BTS_BLL2R := FALSE;
	ELSIF AL_GERAL = TRUE THEN //desliga se alarmes
		SD_BLL2R := FALSE;
		BTS_BLL2R := FALSE;
	END_IF
	
	//Balança liquidos 2 - carga lenta
	IF BTS_BLL2L = TRUE AND SD_BLL2D = FALSE AND AL_GERAL = FALSE THEN
		IF SD_BLL2L = TRUE THEN
			SD_BLL2L := FALSE;
		ELSE
			SD_BLL2L := TRUE;
		END_IF		
		BTS_BLL2L := FALSE;
	ELSIF  AL_GERAL = TRUE THEN //desliga se alarmes
		SD_BLL2L := FALSE;
		BTS_BLL2L := FALSE;
	END_IF

	//Desliga a rosca automaticamente pelo peso
	IF (SD_BLL2L = TRUE OR SD_BLL2R = TRUE) AND LEITURA_PESO_BLL2 > PRST_PESO_BLL2 THEN
		SD_BLL2L := FALSE;
		SD_BLL2R := FALSE;
	END_IF
	
	//Balança liquidos 3 - carga rapida =============================================
	IF BTS_BLL3R = TRUE  AND SD_BLL3D = FALSE AND AL_GERAL = FALSE THEN
		IF SD_BLL3R = TRUE THEN
			SD_BLL3R := FALSE;
		ELSE
			SD_BLL3R := TRUE;
		END_IF		
		BTS_BLL3R := FALSE;		
	ELSIF AL_GERAL = TRUE THEN //desliga se alarmes
		SD_BLL3R := FALSE;
		BTS_BLL3R := FALSE;	
	END_IF

	//Balança liquidos 3 - carga lenta
	IF BTS_BLL3L = TRUE  AND SD_BLL3D = FALSE AND AL_GERAL = FALSE THEN
		IF SD_BLL3L = TRUE THEN
			SD_BLL3L := FALSE;
		ELSE
			SD_BLL3L := TRUE;
		END_IF		
		BTS_BLL3L := FALSE;	
	ELSIF AL_GERAL = TRUE THEN //desliga se alarmes
		SD_BLL3L := FALSE;
		BTS_BLL3L := FALSE;	
	END_IF
	
	//Desliga a rosca automaticamente pelo peso
	IF (SD_BLL3L = TRUE OR SD_BLL3R = TRUE) AND LEITURA_PESO_BLL3 > PRST_PESO_BLL3 THEN
		SD_BLL3L := FALSE;
		SD_BLL3R := FALSE;
	END_IF

	//Balança liquidos 4 - carga rapida =============================================
	IF BTS_BLL4R = TRUE  AND SD_BLL4D = FALSE AND AL_GERAL = FALSE THEN
		IF SD_BLL4R = TRUE THEN
			SD_BLL4R := FALSE;
		ELSE
			SD_BLL4R := TRUE;
		END_IF		
		BTS_BLL4R := FALSE;
	ELSIF  AL_GERAL = TRUE THEN //desliga se alarmes
		SD_BLL4R := FALSE;
		BTS_BLL4R := FALSE;
	END_IF

	//Balança liquidos 4 - carga lenta
	IF BTS_BLL4L = TRUE  AND SD_BLL4D = FALSE AND AL_GERAL = FALSE THEN
		IF SD_BLL4L = TRUE THEN
			SD_BLL4L := FALSE;
		ELSE
			SD_BLL4L := TRUE;
		END_IF		
		BTS_BLL4L := FALSE;	
	ELSIF AL_GERAL = TRUE THEN //desliga se alarmes
		SD_BLL4L := FALSE;
		BTS_BLL4L := FALSE;	
	END_IF
	
	
	//Desliga a rosca automaticamente pelo peso
	IF (SD_BLL4L = TRUE OR SD_BLL4R = TRUE) AND LEITURA_PESO_BLL4 > PRST_PESO_BLL4 THEN
		SD_BLL4L := FALSE;
		SD_BLL4R := FALSE;
	END_IF

	//Descargas das balanças =========================================

	//Balança de sólido 1 - Descarga ====================================
	IF BTS_BLS1D = TRUE  AND AL_GERAL = FALSE  THEN
		IF SD_BLS1 = TRUE THEN			
			SD_BLS1 := FALSE;
		ELSE
			SD_BLS1 := TRUE;
		END_IF		
		BTS_BLS1D:=FALSE;
	ELSIF  AL_GERAL = TRUE  THEN //desliga se alarmes
		SD_BLS1 := FALSE;
		BTS_BLS1D:=FALSE;
	END_IF

	//Balança de sólido 2 - Descarga ====================================
	IF BTS_BLS2D = TRUE  AND AL_GERAL = FALSE  THEN
		IF SD_BLS2 = TRUE THEN
			SD_BLS2 := FALSE;
		ELSE
			SD_BLS2 := TRUE;
		END_IF
		BTS_BLS2D := FALSE;	
	ELSIF  AL_GERAL = TRUE  THEN //desliga se alarmes
		SD_BLS2 := FALSE;
		BTS_BLS2D := FALSE;		
	END_IF

	//Balança de sólido 3 - Descarga ====================================
	IF BTS_BLS3D = TRUE  AND AL_GERAL = FALSE  THEN
		IF SD_BLS3 = TRUE THEN
			SD_BLS3 := FALSE;
		ELSE
			SD_BLS3 := TRUE;
		END_IF
		BTS_BLS3D := FALSE;	
	ELSIF AL_GERAL = TRUE  THEN //desliga se alarmes
		SD_BLS3 := FALSE;
		BTS_BLS3D := FALSE;
	END_IF

	//Balança de sólido 4 - Descarga ====================================
	IF BTS_BLS4D = TRUE  AND AL_GERAL = FALSE THEN
		IF SD_BLS4 = TRUE THEN
			SD_BLS4 := FALSE;
		ELSE
			SD_BLS4 := TRUE;
		END_IF
		BTS_BLS4D := FALSE;	
	ELSIF AL_GERAL = TRUE  THEN //desliga se alarmes
		SD_BLS4 := FALSE;
		BTS_BLS4D := FALSE;	
	END_IF

	//Balança de sólido 5 - Descarga ===================================
	IF BTS_BLS5D = TRUE  AND AL_GERAL = FALSE THEN
		IF SD_BLS5 = TRUE THEN
			SD_BLS5 := FALSE;
		ELSE
			SD_BLS5 := TRUE;
		END_IF
		BTS_BLS5D := FALSE;	
	ELSIF AL_GERAL = TRUE  THEN //desliga se alarmes
		SD_BLS5 := FALSE;	
		BTS_BLS5D := FALSE;
	END_IF

	//Balança de liquido 1 - Descarga ===================================
	IF BTS_BL1D = TRUE  AND AL_GERAL = FALSE  THEN
		IF SD_BLL1D = TRUE THEN
			SD_BLL1D := FALSE;
		ELSE
			SD_BLL1D := TRUE;
		END_IF
		BTS_BL1D := FALSE;	
	ELSIF AL_GERAL = TRUE  THEN //desliga se alarmes
		SD_BLL1D := FALSE;	
		BTS_BL1D := FALSE;
	END_IF

	//Balança de liquido 2 - Descarga ====================================
	IF BTS_BL2D = TRUE AND AL_GERAL = FALSE THEN
		IF SD_BLL2D = TRUE THEN
			SD_BLL2D := FALSE;
		ELSE
			SD_BLL2D := TRUE;
		END_IF	
		BTS_BL2D := FALSE;
	ELSIF AL_GERAL = TRUE THEN //desliga se alarmes
		SD_BLL2D := FALSE;	
		BTS_BL2D := FALSE;
	END_IF

	//Balança de liquido 3 - Descarga ====================================
	IF BTS_BL3D = TRUE AND AL_GERAL = FALSE  THEN
		IF SD_BLL3D = TRUE THEN
			SD_BLL3D := FALSE;
		ELSE
			SD_BLL3D := TRUE;	
		END_IF		
		BTS_BL3D := FALSE;
	ELSIF AL_GERAL = TRUE  THEN //desliga se alarmes
		SD_BLL3D := FALSE;	
		BTS_BL3D := FALSE;
	END_IF

	//Balança de liquido 4 - Descarga ====================================
	IF BTS_BL4D = TRUE  AND AL_GERAL = FALSE  THEN
		IF SD_BLL4D = TRUE THEN
			SD_BLL4D := FALSE;
		ELSE
			SD_BLL4D := TRUE;
		END_IF		
		BTS_BL4D := FALSE;
	ELSIF AL_GERAL = TRUE  THEN //desliga se alarmes
		SD_BLL4D := FALSE;
		BTS_BL4D := FALSE;	
	END_IF	
	

	//Roscas ============================================================

	//Rosca 6 - Horizontal ==============================================
	IF BTS_RC6H = TRUE AND SD_R7 = TRUE AND AL_GERAL = FALSE THEN
		IF SD_R6 = TRUE THEN
			SD_R6 := FALSE;	
		ELSE
			SD_R6 := TRUE;
		END_IF		
		BTS_RC6H := FALSE;	
	ELSIF AL_GERAL = TRUE THEN
		SD_R6 := FALSE;	
		BTS_RC6H := FALSE;	
	END_IF

	//Rosca 7 - Inclinada =================================================
	IF BTS_RC7I = TRUE  AND SD_MXP_P = TRUE AND SD_MXP_T = TRUE AND AL_GERAL = FALSE THEN
		IF SD_R7 = TRUE THEN
			SD_R7 := FALSE;
		ELSE
			SD_R7 := TRUE;
		END_IF		
		BTS_RC7I := FALSE;	
	ELSIF SD_MXP_P = FALSE AND SD_MXP_T = FALSE OR AL_GERAL = TRUE THEN
		SD_R7 := FALSE;
		BTS_RC7I := FALSE;
	END_IF

	
	
	// Aquecimento mexedor principal ****************************		
	
	IF BTS_AQUEMXP = TRUE AND SD_VLMISTURA = FALSE AND AL_GERAL = FALSE THEN
		IF SD_VPMECEDOR =TRUE THEN
			SD_VPMECEDOR := FALSE;
		ELSE
			SD_VPMECEDOR := TRUE;
		END_IF		
		BTS_AQUEMXP := FALSE;	
	ELSIF AL_GERAL = TRUE OR TEMP_VAPOR >= PRST_TEMPE_ALAR_MXP THEN
		SD_VPMECEDOR := FALSE;
		BTS_AQUEMXP := FALSE;
	END_IF
	

	// Bombas ==================================================================
			
	//Bomba de  e Valvula de Agua ======================================
	IF BTS_BAG = TRUE AND AL_GERAL = FALSE  THEN
		IF SD_BAG = TRUE THEN
			SD_BAG := FALSE;
		ELSE
			SD_BAG := TRUE;
		END_IF		
		BTS_BAG := FALSE;	
	ELSIF AL_GERAL = TRUE THEN
		SD_BAG := FALSE;
		BTS_BAG := FALSE;
	END_IF
	
	//Valvula de agua  
	//Liga junto com a bomba de agua
	IF SD_BAG = TRUE THEN
		SD_VLAG := TRUE;
	ELSE
		SD_VLAG := FALSE;
	END_IF
		
	
	//Valvula de saida do misturador principal ================================
	IF BTS_VLSMXP = TRUE AND AL_GERAL = FALSE   THEN
		IF SD_VLMISTURA = TRUE THEN
			SD_VLMISTURA := FALSE;
		ELSE
			SD_VLMISTURA := TRUE;
		END_IF		
		BTS_VLSMXP := FALSE;	
	ELSIF AL_GERAL = TRUE THEN
		SD_VLMISTURA := FALSE;
		BTS_VLSMXP := FALSE;	
	END_IF
	
	
	//Bomba de acusol =================================================================
	PRST_PESO_ACUSOL :=0;
	//Soma peso da BLL4 (Blend) com acusol
	PESO_BLL4_ACUSOL := PRST_PESO_BLL4 + PRST_PESO_ACUSOL;
	

	IF BTS_BACU = TRUE AND AL_GERAL = FALSE  THEN
		IF SD_BACU = TRUE THEN
			SD_VLACU := FALSE;
			SD_BACU := FALSE;			
		ELSE
			SD_BACU := TRUE;
			SD_VLACU := TRUE;
		END_IF		
		BTS_BACU := FALSE;	
	ELSIF AL_GERAL = TRUE OR LEITURA_PESO_BLL4 >= PESO_BLL4_ACUSOL THEN
		SD_VLACU := FALSE;
		SD_BACU := FALSE;
	END_IF	
	
	

	//Comando que devem ser resetado no manual:  ======================================
	
	ST_CICLO_PROCESSO := FALSE;	
	BTS_INICICLO := FALSE;
	CNT_SEQUENCIA_SLURRY := 0;
	INTERVALO_TROCA_SEQUE:= FALSE;
	CONTINUA_SEQUENCIA :=FALSE;
	TRANSFERENCIA_lIBERADA := FALSE;
	ULTIMA_CARGA := FALSE;
	BLS1_CARREGADA := FALSE;
	BLS2_CARREGADA := FALSE;
	BLS3_CARREGADA := FALSE;
	BLS4_CARREGADA := FALSE;
	BLS5_CARREGADA := FALSE;
	BLL1_CARREGADA := FALSE;
	BLL2_CARREGADA := FALSE;
	BLL3_CARREGADA := FALSE;
	BLL4_CARREGADA := FALSE;
ELSE


// Comando automatico ============================================================

	//ciclo ===============================================================
	IF AL_GERAL = FALSE AND BTS_INICICLO = TRUE AND PROGRAMA_CARREGADO_SLURRY = 1 THEN	
		ST_CICLO_PROCESSO := TRUE;			
	END_IF

	//Finaliza ciclo
	IF AL_GERAL = TRUE OR BTS_PARADA_CICLO = TRUE THEN
		BTS_INICICLO := FALSE;
		ST_CICLO_PROCESSO := FALSE;
		INTERVALO_TROCA_SEQUE := FALSE;	
		BTS_PARADA_CICLO :=FALSE;			
	END_IF
	
	//gera pulso inicio de ciclo
	PULSO_INICIO_CICLO(CLK:= ST_CICLO_PROCESSO);
	
	//Carrega o passo 1 ao inicio de ciclo
	IF PULSO_INICIO_CICLO.Q = TRUE THEN
		CNT_SEQUENCIA_SLURRY := 1;
		INTERVALO_TROCA_SEQUE := TRUE;
	END_IF
			

	//Rosca 7 - Inclinada =================================================
	IF (SD_BLS1 = TRUE OR SD_BLS2 = TRUE OR SD_BLS3 = TRUE OR SD_BLS4 = TRUE OR SD_BLS5 = TRUE OR BTS_MASLU = TRUE) AND SD_MXP_T = TRUE THEN		
		SD_R7_AUX := TRUE;
	ELSIF ST_CICLO_PROCESSO = FALSE OR TRANSFERENCIA_lIBERADA = TRUE THEN
		SD_R7_AUX := FALSE;			
	END_IF
		TM_AUX_SD_R7 := ANY_TO_TIME (50000);
		TM_SD_R7 (IN := INICIAR_TEMPO_HOMOGENIZACAO, PT :=  TM_AUX_SD_R7);
		
	IF SD_R7_AUX = TRUE AND SD_BLS5 = TRUE  THEN
		SD_R7 := TRUE;
		ELSIF  TM_SD_R7.Q = TRUE THEN
			
		SD_R7 := FALSE;	
					
	END_IF
	
	//Rosca 6 - Horizontal ==============================================
	IF (SD_BLS1 = TRUE OR SD_BLS2 = TRUE OR SD_BLS3 = TRUE OR SD_BLS4 = TRUE OR SD_BLS5 = TRUE) AND SD_R7 = TRUE THEN		
		SD_R6 := TRUE;
	ELSIF ST_CICLO_PROCESSO = FALSE OR TRANSFERENCIA_lIBERADA = TRUE THEN
		SD_R6 := FALSE;			
	END_IF

	
	//Carga das balanças  ======================================================
	
	// Carga da balanca sólido 1
	//condições: se ciclo + não esta na sequencia + não esta desabilitado + não esta a descarga aberta +
	// peso de leitura menor que preset
	IF  PRST_POSSEQ_BLS1 > 0 AND SD_BLS1 = FALSE AND LEITURA_PESO_BLS1 <= PRST_PESO_BLS1 - 7 AND ULTIMA_BATELADA = FALSE AND FIM_PRODUCAO = FALSE THEN	
		SD_RPO1 := TRUE;
	ELSE
		SD_RPO1 := FALSE;
	END_IF
	IF LEITURA_PESO_BLS1 >= PRST_PESO_BLS1 THEN
		BLS1_CARREGADA := TRUE;
		DESCARGA_INICIADA_BLS1 := FALSE;
	END_IF
	
	
	// Carga da balanca sólido 2
	//condições: se ciclo + não esta na sequencia + não esta desabilitado + não esta a descarga aberta +
	// peso de leitura menor que preset
	IF  PRST_POSSEQ_BLS2 > 0 AND SD_BLS2 = FALSE AND LEITURA_PESO_BLS2 <= PRST_PESO_BLS2 - 7 AND ULTIMA_BATELADA = FALSE AND FIM_PRODUCAO = FALSE THEN	
		SD_RPO2 := TRUE;
	ELSE
		SD_RPO2 := FALSE;
	END_IF
	IF LEITURA_PESO_BLS2 >= PRST_PESO_BLS2 THEN
		BLS2_CARREGADA := TRUE;
		DESCARGA_INICIADA_BLS2 := FALSE;
	END_IF
	
	
	// Carga da balanca sólido 3
	//condições: se ciclo + não esta na sequencia + não esta desabilitado + não esta a descarga aberta +
	// peso de leitura menor que preset
	IF PRST_POSSEQ_BLS3 > 0 AND SD_BLS3 = FALSE AND LEITURA_PESO_BLS3 <= PRST_PESO_BLS3 - 2 AND ULTIMA_BATELADA = FALSE AND FIM_PRODUCAO = FALSE THEN
	
		SD_RPO3 := TRUE;
	ELSE
		SD_RPO3 := FALSE;
	END_IF
	IF LEITURA_PESO_BLS3 >= PRST_PESO_BLS3 - 1 THEN
		BLS3_CARREGADA := TRUE;
		DESCARGA_INICIADA_BLS3 := FALSE;
	END_IF
	
	
	// Carga da balanca sólido 4
	//condições: se ciclo + não esta na sequencia + não esta desabilitado + não esta a descarga aberta +
	// peso de leitura menor que preset
	IF PRST_POSSEQ_BLS4 > 0 AND SD_BLS4 = FALSE AND LEITURA_PESO_BLS4 <= PRST_PESO_BLS4 - 2 AND ULTIMA_BATELADA = FALSE AND FIM_PRODUCAO = FALSE THEN	
		SD_RPO4 := TRUE;
	ELSE
		SD_RPO4 := FALSE;
	END_IF
	IF LEITURA_PESO_BLS4 >= PRST_PESO_BLS4 THEN
		BLS4_CARREGADA := TRUE;
		DESCARGA_INICIADA_BLS4 := FALSE;
	END_IF
	
	
	// Carga da balanca sólido 5
	//condições: se ciclo + não esta na sequencia + não esta desabilitado + não esta a descarga aberta +
	// peso de leitura menor que preset
	IF PRST_POSSEQ_BLS5 > 0 AND SD_BLS5 = FALSE AND LEITURA_PESO_BLS5 <= PRST_PESO_BLS5 - 6 AND ULTIMA_BATELADA = FALSE AND FIM_PRODUCAO = FALSE THEN	
		SD_RPO5 := TRUE;
	ELSE
		SD_RPO5 := FALSE;
	END_IF
	IF LEITURA_PESO_BLS5 >= PRST_PESO_BLS5 THEN
		BLS5_CARREGADA := TRUE;
		DESCARGA_INICIADA_BLS5 := FALSE;
	END_IF
	
	
	// Carga da balanca liquidos 1
	//condições: se ciclo + não esta na sequencia + não esta desabilitado + não esta a descarga aberta +
	// peso de leitura menor que preset
	IF 	PRST_POSSEQ_BLL1 > 0 AND SD_BLL1D = FALSE AND LEITURA_PESO_BLL1 <= PRST_PESO_BLL1 AND ULTIMA_BATELADA = FALSE AND FIM_PRODUCAO = FALSE THEN	
	
		//se peso real estiver faltando 5kg para chegar no preset, desliga valvula rapida para precisão		
		IF LEITURA_PESO_BLL1 >= PRST_PESO_BLL1 - 16 THEN
			SD_BLL1R := FALSE;
		ELSE
			SD_BLL1R := TRUE;
		END_IF
		
		IF LEITURA_PESO_BLL1 >= PRST_PESO_BLL1 - 1 THEN
			SD_BLL1L := FALSE;
		ELSE
			SD_BLL1L := TRUE;
		END_IF
		//SD_BLL1L := TRUE;
		
	ELSE
		SD_BLL1R := FALSE;
		SD_BLL1L := FALSE;
	END_IF
	IF LEITURA_PESO_BLL1 >= PRST_PESO_BLL1 - 2 THEN
		BLL1_CARREGADA := TRUE;
		DESCARGA_INICIADA_BLL1 := FALSE;
	END_IF
	
	
	// Carga da balanca liquidos 2
	//condições: se ciclo + não esta na sequencia + não esta desabilitado + não esta a descarga aberta +
	// peso de leitura menor que preset
	IF PRST_POSSEQ_BLL2 > 0 AND SD_BLL2D = FALSE AND LEITURA_PESO_BLL2 <= PRST_PESO_BLL2 AND ULTIMA_BATELADA = FALSE AND FIM_PRODUCAO = FALSE THEN
		
		//se peso real estiver faltando 5kg para chegar no preset, desliga valvula rapida para precisão		
		IF LEITURA_PESO_BLL2 >= PRST_PESO_BLL2 - 10 THEN
			SD_BLL2R := FALSE;
		ELSE
			SD_BLL2R := TRUE;
		END_IF
		
IF LEITURA_PESO_BLL2 >= PRST_PESO_BLL2 - 1 THEN
			SD_BLL2L := FALSE;
		ELSE
			SD_BLL2L := TRUE;
		END_IF
		//SD_BLL2L := TRUE;
		
	ELSE
		SD_BLL2R := FALSE;
		SD_BLL2L := FALSE;
	END_IF
	IF LEITURA_PESO_BLL2 >= PRST_PESO_BLL2 - 3 THEN
		BLL2_CARREGADA := TRUE;
		DESCARGA_INICIADA_BLL2 := FALSE;
	END_IF
	
	
	// Carga da balanca liquidos 3
	//condições: se ciclo + não esta na sequencia + não esta desabilitado + não esta a descarga aberta +
	// peso de leitura menor que preset
	IF PRST_POSSEQ_BLL3 > 0 AND SD_BLL3D = FALSE AND LEITURA_PESO_BLL3 <= PRST_PESO_BLL3 AND ULTIMA_BATELADA = FALSE AND FIM_PRODUCAO = FALSE THEN
		
		//se peso real estiver faltando 5kg para chegar no preset, desliga valvula rapida para precisão		
		IF LEITURA_PESO_BLL3 >= PRST_PESO_BLL3 - 10 THEN
			SD_BLL3R := FALSE;
		ELSE
			SD_BLL3R := TRUE;
		END_IF
		
		SD_BLL3L := TRUE;
		
	ELSE
		SD_BLL3R := FALSE;
		SD_BLL3L := FALSE;
	END_IF
	IF LEITURA_PESO_BLL3 >= PRST_PESO_BLL3 THEN
		BLL3_CARREGADA := TRUE;
		DESCARGA_INICIADA_BLL3 := FALSE;
	END_IF
	
	
	// Carga da balanca liquidos 4
	//condições: se ciclo + não esta na sequencia + não esta desabilitado + não esta a descarga aberta +
	// peso de leitura menor que preset
	IF 	PRST_POSSEQ_BLL4 > 0 AND SD_BLL4D = FALSE AND LEITURA_PESO_BLL4 <= PRST_PESO_BLL4 AND ULTIMA_BATELADA = FALSE AND FIM_PRODUCAO = FALSE THEN
						
		//se peso real estiver faltando 5kg para chegar no preset, desliga valvula rapida para precisão		
		IF LEITURA_PESO_BLL4 >= PRST_PESO_BLL4 - 5 THEN
			SD_BLL4R := FALSE;
		ELSE
			SD_BLL4R := TRUE;
		END_IF
		
		SD_BLL4L := TRUE;
		
	ELSE
		SD_BLL4R := FALSE;
		SD_BLL4L := FALSE;
	END_IF
	
	
	//carrega o acusol depois do blend
	
	//Soma peso da BLL4 (Blend) com acusol
	PESO_BLL4_ACUSOL := PRST_PESO_BLL4 + PRST_PESO_ACUSOL;
	
	IF LEITURA_PESO_BLL4 >= PRST_PESO_BLL4 AND LEITURA_PESO_BLL4 < PESO_BLL4_ACUSOL  THEN
		SD_BACU := TRUE;
		SD_VLACU := TRUE;
	ELSE
		SD_BACU := FALSE;
		SD_VLACU := FALSE;
	END_IF
	IF LEITURA_PESO_BLL4 >= PESO_BLL4_ACUSOL THEN
		BLL4_CARREGADA := TRUE;
		DESCARGA_INICIADA_BLL4 := FALSE;
	END_IF
	
	
	//ciclo dos equipamentos ==========================================================
	
	
	// Descarga das balanças 
		
	//Descarga Balança sólido 1 ============================================
	//Condições: Em ciclo + sem alarmes + na sequencia correta + estar habilitado + BL carregada + valvula saida MXP fechada + 
	//roscas 6 e 7 ligadas + misturador ligado + sem alarme geral
	//Senão se:
	// Em ciclo + (se descarga ligada e balança descarregada) + na sequencia + 
	// sem alarme geral
	
	IF ST_CICLO_PROCESSO = TRUE  AND PRST_POSSEQ_BLS1 = CNT_SEQUENCIA_SLURRY AND PRST_POSSEQ_BLS1 > 0 AND SD_VLMISTURA = FALSE 
	AND BLS1_CARREGADA = TRUE  AND ST_CFMXP = TRUE AND AL_GERAL = FALSE  AND CONTINUA_SEQUENCIA = TRUE AND (LEITURA_PESO_BLS1 >= PRST_PESO_BLS1 OR BTS_PERMI_DESCAR_PESO_MAX_BLS1 = TRUE) 
	AND DESCARGA_INICIADA_BLS1 = FALSE THEN	
		
		SD_BLS1 := TRUE;	
		DESCARGA_INICIADA_BLS1 := TRUE;
		
	ELSIF ST_CICLO_PROCESSO = TRUE  AND (SD_BLS1 = TRUE AND LEITURA_PESO_BLS1 < PRST_ZERO_PESO_BLS1) 
	AND PRST_POSSEQ_BLS1 = CNT_SEQUENCIA_SLURRY AND AL_GERAL = FALSE THEN
		
		SD_BLS1 := FALSE;
		CNT_SEQUENCIA_SLURRY := CNT_SEQUENCIA_SLURRY + 1; //incrementa a sequencia
		INTERVALO_TROCA_SEQUE := TRUE; 					 // ativa retardo de inicio da sequencia, para limpar as roscas
		CONTINUA_SEQUENCIA:= FALSE;
		BLS1_CARREGADA := FALSE;
		BTS_PERMI_DESCAR_PESO_MAX_BLS1 := FALSE;
		DESCARGA_INICIADA_BLS1 := FALSE;
	ELSIF ST_CICLO_PROCESSO = FALSE THEN		
		
		SD_BLS1 := FALSE;
	END_IF
	

	//Descarga Balança sólido 2 ============================================	
	//Condições: Em ciclo + sem alarmes + na sequencia correta + estar habilitado +  BL carregada + valvula saida MXP fechada + 
	//roscas 6 e 7 ligadas + misturador ligado + sem alarme geral	
	//Senão se:
	// Em ciclo + (se descarga ligada e balança descarregada) + na sequencia + 
	// sem alarme geral
	
	IF ST_CICLO_PROCESSO = TRUE  AND PRST_POSSEQ_BLS2 = CNT_SEQUENCIA_SLURRY AND PRST_POSSEQ_BLS2 > 0 AND SD_VLMISTURA = FALSE
	AND BLS2_CARREGADA = TRUE AND ST_CFMXP = TRUE AND AL_GERAL = FALSE AND  CONTINUA_SEQUENCIA = TRUE AND (LEITURA_PESO_BLS2 >= PRST_PESO_BLS2 OR BTS_PERMI_DESCAR_PESO_MAX_BLS2 = TRUE) 
	AND DESCARGA_INICIADA_BLS2 = FALSE THEN	
		
		SD_BLS2 := TRUE;	
		DESCARGA_INICIADA_BLS2 := TRUE;
		
	ELSIF ST_CICLO_PROCESSO = TRUE AND (SD_BLS2 = TRUE AND LEITURA_PESO_BLS2 < PRST_ZERO_PESO_BLS2) 
	AND PRST_POSSEQ_BLS2 = CNT_SEQUENCIA_SLURRY AND AL_GERAL = FALSE THEN
		
		SD_BLS2 := FALSE;
		CNT_SEQUENCIA_SLURRY := CNT_SEQUENCIA_SLURRY + 1; //incrementa a sequencia
		INTERVALO_TROCA_SEQUE := TRUE; 					 // ativa retardo de inicio da sequencia, para limpar as roscas
		CONTINUA_SEQUENCIA := FALSE;
		BTS_PERMI_DESCAR_PESO_MAX_BLS2 := FALSE;
		BLS2_CARREGADA := FALSE;
		DESCARGA_INICIADA_BLS2 := FALSE;
	ELSIF ST_CICLO_PROCESSO = FALSE THEN		
		
		SD_BLS2 := FALSE;
	END_IF
		
	//Descarga Balança sólido 3 ============================================
	//Condições: Em ciclo + sem alarmes + na sequencia correta + estar habilitado +  BL carregada + valvula saida MXP fechada + 
	//roscas 6 e 7 ligadas + misturador ligado + sem alarme geral	
	//Senão se:
	// Em ciclo + (se descarga ligada e balança descarregada) + na sequencia + 
	// sem alarme geral
	
	IF ST_CICLO_PROCESSO = TRUE AND PRST_POSSEQ_BLS3 = CNT_SEQUENCIA_SLURRY AND  PRST_POSSEQ_BLS3 > 0 AND SD_VLMISTURA = FALSE
	AND BLS3_CARREGADA = TRUE  AND ST_CFMXP = TRUE AND AL_GERAL = FALSE AND  CONTINUA_SEQUENCIA = TRUE AND (LEITURA_PESO_BLS3 >= PRST_PESO_BLS3 OR BTS_PERMI_DESCAR_PESO_MAX_BLS3 = TRUE) 
	AND DESCARGA_INICIADA_BLS3 = FALSE THEN	
		
		SD_BLS3 := TRUE;	
		DESCARGA_INICIADA_BLS3 := TRUE;
		
	ELSIF ST_CICLO_PROCESSO = TRUE AND (SD_BLS3 = TRUE AND LEITURA_PESO_BLS3 < PRST_ZERO_PESO_BLS3) 
	AND PRST_POSSEQ_BLS3 = CNT_SEQUENCIA_SLURRY AND AL_GERAL = FALSE THEN
		
		SD_BLS3 := FALSE;
		CNT_SEQUENCIA_SLURRY := CNT_SEQUENCIA_SLURRY + 1; //incrementa a sequencia
		INTERVALO_TROCA_SEQUE := TRUE; 					 // ativa retardo de inicio da sequencia, para limpar as roscas
		CONTINUA_SEQUENCIA := FALSE;
		BTS_PERMI_DESCAR_PESO_MAX_BLS3 := FALSE;
		BLS3_CARREGADA := FALSE;
		DESCARGA_INICIADA_BLS3 := FALSE;
	ELSIF ST_CICLO_PROCESSO = FALSE THEN		
		
		SD_BLS3 := FALSE;
	END_IF
		
	//Descarga Balança sólido 4 ============================================	
	//Condições: Em ciclo + sem alarmes + na sequencia correta + estar habilitado +  BL carregada + valvula saida MXP fechada + 
	//roscas 6 e 7 ligadas + misturador ligado + sem alarme geral
	//Senão se:
	// Em ciclo + (se descarga ligada e balança descarregada) + na sequencia + 
	// sem alarme geral
	
	IF ST_CICLO_PROCESSO = TRUE AND PRST_POSSEQ_BLS4 = CNT_SEQUENCIA_SLURRY AND PRST_POSSEQ_BLS4 > 0 AND SD_VLMISTURA = FALSE
	AND BLS4_CARREGADA = TRUE  AND ST_CFMXP = TRUE AND AL_GERAL = FALSE AND  CONTINUA_SEQUENCIA = TRUE AND (LEITURA_PESO_BLS4 >= (PRST_PESO_BLS4 - 3) OR BTS_PERMI_DESCAR_PESO_MAX_BLS4 = TRUE) 
	AND DESCARGA_INICIADA_BLS4 = FALSE THEN	
		
		SD_BLS4 := TRUE;
		DESCARGA_INICIADA_BLS4 := TRUE;	
		
	ELSIF ST_CICLO_PROCESSO = TRUE AND (SD_BLS4 = TRUE AND LEITURA_PESO_BLS4 < PRST_ZERO_PESO_BLS4) 
	AND PRST_POSSEQ_BLS4 = CNT_SEQUENCIA_SLURRY AND AL_GERAL = FALSE THEN
		
		SD_BLS4 := FALSE;
		CNT_SEQUENCIA_SLURRY := CNT_SEQUENCIA_SLURRY + 1; //incrementa a sequencia
		INTERVALO_TROCA_SEQUE := TRUE; 					 // ativa retardo de inicio da sequencia, para limpar as roscas
		CONTINUA_SEQUENCIA := FALSE;
		BTS_PERMI_DESCAR_PESO_MAX_BLS4 := FALSE;
		BLS4_CARREGADA := FALSE;
		DESCARGA_INICIADA_BLS4 := FALSE;	
	ELSIF ST_CICLO_PROCESSO = FALSE THEN		
		
		SD_BLS4 := FALSE;
	END_IF
	
	//Descarga Balança sólido 5 ============================================	
	//Condições: Em ciclo + sem alarmes + na sequencia correta + estar habilitado +  BL carregada + valvula saida MXP fechada + 
	//roscas 6 e 7 ligadas + misturador ligado + sem alarme geral
	//Senão se:
	// Em ciclo + (se descarga ligada e balança descarregada) + na sequencia + 
	// sem alarme geral
	
	IF ST_CICLO_PROCESSO = TRUE AND PRST_POSSEQ_BLS5 = CNT_SEQUENCIA_SLURRY AND  PRST_POSSEQ_BLS5 > 0 AND SD_VLMISTURA = FALSE
	AND BLS5_CARREGADA = TRUE  AND ST_CFMXP = TRUE AND AL_GERAL = FALSE AND  CONTINUA_SEQUENCIA = TRUE AND (LEITURA_PESO_BLS5 >= (PRST_PESO_BLS5 - 3) OR BTS_PERMI_DESCAR_PESO_MAX_BLS5 = TRUE) 
	AND DESCARGA_INICIADA_BLS5 = FALSE THEN	
		
		SD_BLS5 := TRUE;
		DESCARGA_INICIADA_BLS5 := TRUE;	
		
	ELSIF ST_CICLO_PROCESSO = TRUE AND (SD_BLS5 = TRUE AND LEITURA_PESO_BLS5 < PRST_ZERO_PESO_BLS5) 
	AND PRST_POSSEQ_BLS5 = CNT_SEQUENCIA_SLURRY AND AL_GERAL = FALSE THEN
		
		SD_BLS5 := FALSE;
		CNT_SEQUENCIA_SLURRY := CNT_SEQUENCIA_SLURRY + 1; //incrementa a sequencia
		INTERVALO_TROCA_SEQUE := TRUE; 					 // ativa retardo de inicio da sequencia, para limpar as roscas
		CONTINUA_SEQUENCIA := FALSE;
		BTS_PERMI_DESCAR_PESO_MAX_BLS5 := FALSE;
		BLS5_CARREGADA := FALSE;
		DESCARGA_INICIADA_BLS5 := FALSE;
	ELSIF ST_CICLO_PROCESSO = FALSE THEN
		
		SD_BLS5 := FALSE;
	END_IF
	
	
	//Descarga Balança liquido 1 ============================================
	//Condições: Em ciclo +  na sequencia correta + estar habilitado + BL carregada +
	//misturador ligado + sem alarme geral + valvula saida MXP fechada 
	//Senão se:
	// Em ciclo + (se descarga ligada e balança descarregada) + na sequencia + 
	// sem alarme geral
	
	IF ST_CICLO_PROCESSO = TRUE AND PRST_POSSEQ_BLL1 = CNT_SEQUENCIA_SLURRY AND  PRST_POSSEQ_BLL1 > 0 
	AND BLL1_CARREGADA = TRUE AND ST_CFMXP = TRUE AND AL_GERAL = FALSE AND SD_VLMISTURA = FALSE AND CONTINUA_SEQUENCIA = TRUE 
	AND (LEITURA_PESO_BLL1 >= PRST_PESO_BLL1 OR BTS_PERMI_DESCAR_PESO_MAX_BLL1 = TRUE) AND DESCARGA_INICIADA_BLL1 = FALSE THEN
		
		SD_BLL1D := TRUE;	
		DESCARGA_INICIADA_BLL1 := TRUE;
	
	ELSIF ST_CICLO_PROCESSO = TRUE  AND (SD_BLL1D = TRUE AND LEITURA_PESO_BLL1 < PRST_ZERO_PESO_BLL1) 
	AND PRST_POSSEQ_BLL1 = CNT_SEQUENCIA_SLURRY AND AL_GERAL = FALSE THEN
	
		SD_BLL1D := FALSE;
		CNT_SEQUENCIA_SLURRY := CNT_SEQUENCIA_SLURRY + 1; //incrementa a sequencia
		INTERVALO_TROCA_SEQUE := TRUE; 					 // ativa retardo de inicio da sequencia, para limpar as roscas
		CONTINUA_SEQUENCIA := FALSE;
		BTS_PERMI_DESCAR_PESO_MAX_BLL1 := FALSE;
		BLL1_CARREGADA:= FALSE;
		DESCARGA_INICIADA_BLL1 := FALSE;
	ELSIF ST_CICLO_PROCESSO = FALSE THEN
		SD_BLL1D := FALSE;
	END_IF
	
	
	//Descarga Balança liquido 2 ============================================
	//Condições: Em ciclo +  na sequencia correta + estar habilitado + BL carregada +
	//misturador ligado + sem alarme geral + valvula saida MXP fechada 
	//Senão se:
	// Em ciclo + (se descarga ligada e balança descarregada) + na sequencia + 
	// sem alarme geral
	
	IF ST_CICLO_PROCESSO = TRUE AND PRST_POSSEQ_BLL2 = CNT_SEQUENCIA_SLURRY AND  PRST_POSSEQ_BLL2 > 0 
	AND BLL2_CARREGADA = TRUE AND ST_CFMXP = TRUE AND AL_GERAL = FALSE AND SD_VLMISTURA = FALSE AND  CONTINUA_SEQUENCIA = TRUE 
	AND (LEITURA_PESO_BLL2 >= PRST_PESO_BLL2 OR BTS_PERMI_DESCAR_PESO_MAX_BLL2 = TRUE) AND DESCARGA_INICIADA_BLL2 = FALSE THEN
		
		SD_BLL2D := TRUE;
		DESCARGA_INICIADA_BLL2 := TRUE;
		
	ELSIF ST_CICLO_PROCESSO = TRUE  AND (SD_BLL2D = TRUE AND LEITURA_PESO_BLL2 < PRST_ZERO_PESO_BLL2) 
	AND PRST_POSSEQ_BLL2 = CNT_SEQUENCIA_SLURRY AND AL_GERAL = FALSE THEN
	
		SD_BLL2D := FALSE;
		CNT_SEQUENCIA_SLURRY := CNT_SEQUENCIA_SLURRY + 1; //incrementa a sequencia
		INTERVALO_TROCA_SEQUE := TRUE; 					 // ativa retardo de inicio da sequencia, para limpar as roscas
		CONTINUA_SEQUENCIA := FALSE;
		BTS_PERMI_DESCAR_PESO_MAX_BLL2 := FALSE;
		BLL2_CARREGADA:= FALSE;
		DESCARGA_INICIADA_BLL2 := FALSE;
	ELSIF ST_CICLO_PROCESSO = FALSE THEN
		SD_BLL2D := FALSE;
	END_IF
	
	
	//Descarga Balança liquido 3 ============================================
	//Condições: Em ciclo +  na sequencia correta + estar habilitado + BL carregada +
	//misturador ligado + sem alarme geral + valvula saida MXP fechada 
	//Senão se:
	// Em ciclo + (se descarga ligada e balança descarregada) + na sequencia + 
	// sem alarme geral
	
	IF ST_CICLO_PROCESSO = TRUE AND PRST_POSSEQ_BLL3 = CNT_SEQUENCIA_SLURRY AND  PRST_POSSEQ_BLL3 > 0 
	AND BLL3_CARREGADA = TRUE AND ST_CFMXP = TRUE AND AL_GERAL = FALSE AND SD_VLMISTURA = FALSE AND CONTINUA_SEQUENCIA = TRUE 
	AND (LEITURA_PESO_BLL3 >= PRST_PESO_BLL3 OR BTS_PERMI_DESCAR_PESO_MAX_BLL3 = TRUE) AND DESCARGA_INICIADA_BLL3 = FALSE THEN
		
		SD_BLL3D := TRUE;
		DESCARGA_INICIADA_BLL3 := TRUE;
	
	ELSIF ST_CICLO_PROCESSO = TRUE  AND (SD_BLL3D = TRUE AND LEITURA_PESO_BLL3 < PRST_ZERO_PESO_BLL3) 
	AND PRST_POSSEQ_BLL3 = CNT_SEQUENCIA_SLURRY AND AL_GERAL = FALSE THEN
	
		SD_BLL3D := FALSE;
		CNT_SEQUENCIA_SLURRY := CNT_SEQUENCIA_SLURRY + 1; //incrementa a sequencia
		INTERVALO_TROCA_SEQUE := TRUE; 					 // ativa retardo de inicio da sequencia, para limpar as roscas
		CONTINUA_SEQUENCIA := FALSE;
		BTS_PERMI_DESCAR_PESO_MAX_BLL3 := FALSE;
		BLL3_CARREGADA:= FALSE;
		DESCARGA_INICIADA_BLL3 := FALSE;
	ELSIF ST_CICLO_PROCESSO = FALSE THEN
		SD_BLL3D := FALSE;
	END_IF
	
	
	//Descarga Balança liquido 4 ============================================
	//Condições: Em ciclo +  na sequencia correta + estar habilitado + BL carregada +
	//misturador ligado + sem alarme geral + valvula saida MXP fechada 
	//Senão se:
	// Em ciclo + (se descarga ligada e balança descarregada) + na sequencia + 
	// sem alarme geral
	
	IF ST_CICLO_PROCESSO = TRUE AND PRST_POSSEQ_BLL4 = CNT_SEQUENCIA_SLURRY AND PRST_POSSEQ_BLL4 > 0 
	AND BLL4_CARREGADA = TRUE AND ST_CFMXP = TRUE AND AL_GERAL = FALSE AND SD_VLMISTURA = FALSE AND CONTINUA_SEQUENCIA = TRUE 
	AND (LEITURA_PESO_BLL4 >= PRST_PESO_BLL4 OR BTS_PERMI_DESCAR_PESO_MAX_BLL4 = TRUE) AND DESCARGA_INICIADA_BLL4 = FALSE THEN
		
		SD_BLL4D := TRUE;
		DESCARGA_INICIADA_BLL4 := TRUE;
		
	ELSIF ST_CICLO_PROCESSO = TRUE  AND (SD_BLL4D = TRUE AND LEITURA_PESO_BLL4 < PRST_ZERO_PESO_BLL4) 
	AND PRST_POSSEQ_BLL4 = CNT_SEQUENCIA_SLURRY AND AL_GERAL = FALSE THEN
	
		SD_BLL4D := FALSE;
		CNT_SEQUENCIA_SLURRY := CNT_SEQUENCIA_SLURRY + 1; //incrementa a sequencia
		INTERVALO_TROCA_SEQUE := TRUE; 					 // ativa retardo de inicio da sequencia, para limpar as roscas
		CONTINUA_SEQUENCIA := FALSE;
		BTS_PERMI_DESCAR_PESO_MAX_BLL4 := FALSE;
		BLL4_CARREGADA:= FALSE;
		DESCARGA_INICIADA_BLL4 := FALSE;
	ELSIF ST_CICLO_PROCESSO = FALSE THEN
		SD_BLL4D := FALSE;
	END_IF
	
	
	//Tempo reação ======================================================
	
	//multiplica o tempo de reação por 1000, por ser base de tempo em milisegundos
	TEMPO_REACAO_TEMPORARIO := PRST_TEMPO_REACAO * 1000;	
	//converte para time
	TEMPO_REACAO:= ANY_TO_TIME(TEMPO_REACAO_TEMPORARIO);
	
	IF ST_CICLO_PROCESSO = TRUE AND PRST_POSSEQ_TEMPO_REACAO = CNT_SEQUENCIA_SLURRY AND AL_GERAL = FALSE AND CONTINUA_SEQUENCIA =TRUE THEN
		INICIAR_TEMPO_REACAO := TRUE;
	ELSE
		INICIAR_TEMPO_REACAO := FALSE;
	END_IF

	//conta tempo de reação
	TMR_REACAO(IN:=INICIAR_TEMPO_REACAO,PT:=TEMPO_REACAO);
	
	IF TMR_REACAO.Q = TRUE THEN
		INICIAR_TEMPO_REACAO := FALSE;
		CNT_SEQUENCIA_SLURRY := CNT_SEQUENCIA_SLURRY + 1; //incrementa a sequencia
		INTERVALO_TROCA_SEQUE := TRUE; 					 // ativa retardo de inicio da sequencia, para limpar as roscas
		CONTINUA_SEQUENCIA := FALSE;
	END_IF
	
	
	//Tempo hidratação ======================================================
	
	//multiplica o tempo de hidratação por 1000, por ser base de tempo em milisegundos
	TEMPO_HIDRATA_TEMPORARIO := PRST_TEMPO_HIDRATACAO * 1000;	
	//converte para time
	TEMPO_HIDRATA:= ANY_TO_TIME(TEMPO_HIDRATA_TEMPORARIO);
	
	IF ST_CICLO_PROCESSO = TRUE AND PRST_POSSEQ_TEMPO_HIDRATA = CNT_SEQUENCIA_SLURRY AND AL_GERAL = FALSE AND CONTINUA_SEQUENCIA = TRUE THEN
		INICIAR_TEMPO_HIDRATACAO := TRUE;
	ELSE
		INICIAR_TEMPO_HIDRATACAO := FALSE;
	END_IF

	//conta tempo de hidratacao
	TMR_HIDRATA(IN:=INICIAR_TEMPO_HIDRATACAO,PT:=TEMPO_HIDRATA);
	
	IF TMR_HIDRATA.Q = TRUE THEN
		INICIAR_TEMPO_HIDRATACAO := FALSE;
		CNT_SEQUENCIA_SLURRY := CNT_SEQUENCIA_SLURRY + 1; //incrementa a sequencia
		INTERVALO_TROCA_SEQUE := TRUE; 					 // ativa retardo de inicio da sequencia, para limpar as roscas
		CONTINUA_SEQUENCIA := FALSE;
	END_IF
	
	
	//Tempo Homogenização ======================================================
	
	//multiplica o tempo de hidratação por 1000, por ser base de tempo em milisegundos
	TEMPO_HOMOGE_TEMPORARIO := PRST_TEMPO_HOMOGENIZACAO * 1000;	
	//converte para time
	TEMPO_HOMOGE:= ANY_TO_TIME(TEMPO_HOMOGE_TEMPORARIO);
	
	IF ST_CICLO_PROCESSO = TRUE AND PRST_POSSEQ_TEMPO_HOMOGE = CNT_SEQUENCIA_SLURRY AND AL_GERAL = FALSE AND CONTINUA_SEQUENCIA = TRUE THEN
		INICIAR_TEMPO_HOMOGENIZACAO := TRUE;
	ELSE
		INICIAR_TEMPO_HOMOGENIZACAO := FALSE;
	END_IF

	//conta tempo de homogenização
	TMR_HOMOGE(IN:=INICIAR_TEMPO_HOMOGENIZACAO,PT:=TEMPO_HOMOGE);
	
	IF TMR_HOMOGE.Q = TRUE THEN
		INICIAR_TEMPO_HOMOGENIZACAO := FALSE;
		CNT_SEQUENCIA_SLURRY := CNT_SEQUENCIA_SLURRY + 1; //incrementa a sequencia
		INTERVALO_TROCA_SEQUE := TRUE; 					 // ativa retardo de inicio da sequencia, para limpar as roscas
		CONTINUA_SEQUENCIA :=FALSE;
	END_IF
	
	
	//Agua ============================================================================
	
	IF ST_CICLO_PROCESSO = TRUE AND PRST_POSSEQ_AGUA = CNT_SEQUENCIA_SLURRY AND AL_GERAL = FALSE AND CONTINUA_SEQUENCIA = TRUE AND AGUA_DOSADA = FALSE THEN
		SD_BAG := TRUE;
		SD_VLAG := TRUE;
	ELSE
		SD_BAG := FALSE;	
		SD_VLAG := FALSE;	
	END_IF 
	
	
	
	//Vapor ============================================================================
	
	//liga controle de temperatura entre minimo e maximo
	IF ST_CICLO_PROCESSO = TRUE AND PRST_POSSEQ_VAPOR = CNT_SEQUENCIA_SLURRY AND AL_GERAL = FALSE AND CONTINUA_SEQUENCIA = TRUE THEN
		LIGA_CONTROLE_TEMPERATURA_MXP := TRUE;	
		//CNT_SEQUENCIA_SLURRY := CNT_SEQUENCIA_SLURRY + 1; //incrementa a sequencia
		//INTERVALO_TROCA_SEQUE := TRUE; 					 // ativa retardo de inicio da sequencia, para limpar as roscas		
		//CONTINUA_SEQUENCIA :=FALSE;	
	END_IF
	//Desliga controle de temperatura entre minimo e maximo
	IF ST_CICLO_PROCESSO = FALSE THEN
		LIGA_CONTROLE_TEMPERATURA_MXP := FALSE;
	END_IF
	
	//liga valvula de vapor
	IF LIGA_CONTROLE_TEMPERATURA_MXP = TRUE AND TEMP_VAPOR <= PRST_TEMPE_MIN_MXP AND TEMP_VAPOR < PRST_TEMPE_ALAR_MXP  THEN		
		SD_VPMECEDOR := TRUE;				
	END_IF
	
	//Desliga valvula de vapor
	
	IF LIGA_CONTROLE_TEMPERATURA_MXP = FALSE OR TEMP_VAPOR >= PRST_TEMPE_MAX_MXP THEN
		SD_VPMECEDOR := FALSE;
	END_IF
 	
	//TEMP_VAPOR >= PRST_TEMPE_ALAR_MXP Adicionado 06/02/22=====ROBY=====
		IF 	TEMP_VAPOR >= PRST_TEMPE_ALAR_MXP  THEN
		SD_VPMECEDOR := FALSE;
	END_IF
	
	//Libera valvula saida do misturador e a fase de Transferencia ======================
	//deliga vapor
	IF ST_CICLO_PROCESSO = TRUE AND PRST_POSSEQ_VALSAIDA_MXP = CNT_SEQUENCIA_SLURRY AND AL_GERAL = FALSE AND CONTINUA_SEQUENCIA = TRUE THEN
		TRANSFERENCIA_lIBERADA := TRUE;
		LIGA_CONTROLE_TEMPERATURA_MXP := FALSE;	
		RESET_AGUA_AUTO := TRUE;		
	END_IF
	
	//valvula saida do misturador Principal
	IF ST_CICLO_PROCESSO = TRUE AND TRANSFERENCIA_lIBERADA = TRUE AND SD_BBTRANS = TRUE THEN
		SD_VLMISTURA :=TRUE;
	ELSE
		SD_VLMISTURA := FALSE;
	END_IF
	
	//transferencia concluida
	IF TRANSFERENCIA_lIBERADA = TRUE AND LEITURA_NI_MISTPRIN < PRST_NIVEL_MINIMO_MPX THEN
		TRANSFERENCIA_lIBERADA := FALSE;
		LEITURA_BATELADA_ATUAL := LEITURA_BATELADA_ATUAL + 1;
		LEITURA_BATELADA_TOTAL := LEITURA_BATELADA_TOTAL + 1;
		INTERVALO_TROCA_SEQUE := TRUE;
		CNT_SEQUENCIA_SLURRY := 0;			
	END_IF
	
	VAL_REG_PESO_MSP := INICIAR_TEMPO_HOMOGENIZACAO; //SET PARA REGISTRA HISTORICO DE PESO DO MISTURADOR
	
	
	//Retardo troca de sequencia ========================================================
	
	//tempo de intervalo troca de numero sequencia	
	TMR_TROCA_SEQUENCIA(IN:=INTERVALO_TROCA_SEQUE,PT:=T#5S);
	//habilita continuidade da sequencia
	IF TMR_TROCA_SEQUENCIA.Q = TRUE THEN
		CONTINUA_SEQUENCIA := TRUE;
		INTERVALO_TROCA_SEQUE := FALSE;
	END_IF
	
	//Bloqueia a carga ds balanças =====================================================
	
	//Ultima carga
	IF BTS_ULTIMA_CARGA = TRUE AND ST_CICLO_PROCESSO = TRUE THEN
		IF ULTIMA_CARGA = TRUE THEN
			ULTIMA_CARGA := FALSE;
		ELSE
			ULTIMA_CARGA :=TRUE;
		END_IF
		BTS_ULTIMA_CARGA := FALSE;
	END_IF
	//desliga em caso de alarme
	IF AL_GERAL = TRUE OR ST_CICLO_PROCESSO = FALSE THEN
		ULTIMA_CARGA := FALSE;
	END_IF
	
	//Ultima batelada, bloqueia a carga de materiais
	IF (LEITURA_BATELADA_ATUAL >= PRST_QNT_BATELADAS - 1 AND ST_CICLO_PROCESSO = TRUE) OR ULTIMA_CARGA = TRUE THEN
		ULTIMA_BATELADA := TRUE;
	ELSE
		ULTIMA_BATELADA := FALSE;
	END_IF
	
	
	//Verifica a quantidade de batelada, termina ciclo  ================================
	IF LEITURA_BATELADA_ATUAL >= PRST_QNT_BATELADAS THEN
		ST_CICLO_PROCESSO := FALSE;
		CNT_SEQUENCIA_SLURRY := 0;
		LEITURA_BATELADA_ATUAL := 0;
		//ULTIMA_BATELADA := FALSE;
	END_IF
	
	//Comandos que devem ser resetados no automatico
	BTS_RPO1 := FALSE;
	BTS_RPO2 := FALSE;
	BTS_RPO3 := FALSE;
	BTS_RPO4 := FALSE;
	BTS_RPO5 := FALSE;
	BTS_BLL1L := FALSE;
	BTS_BLL2L := FALSE;
	BTS_BLL3L := FALSE;
	BTS_BLL4L := FALSE;
	BTS_BLL1R := FALSE;
	BTS_BLL2R := FALSE;
	BTS_BLL3R := FALSE;
	BTS_BLL4R := FALSE;
	
	
END_IF  // final do manual/automatico ========================================================================


//Comandos que não dependem do manual/automatico ==================================

//Mexedor principal =====================================================
	
	IF BTS_CFMXP = TRUE AND AL_GERAL = FALSE THEN
		IF LIGA_MEXEDOR = TRUE THEN
			LIGA_MEXEDOR := FALSE;
		ELSE
			LIGA_MEXEDOR := TRUE;
		END_IF		
		BTS_CFMXP := FALSE;
	ELSIF AL_GERAL = TRUE THEN
		LIGA_MEXEDOR := FALSE;	
	END_IF
	
	//comando estrela
	//LIGA ESTRELA	
	IF LIGA_MEXEDOR = TRUE  THEN
		IF LIGA_ESTRELA_MXP = FALSE THEN
			//Contatora estrela
			SD_MXP_E := TRUE;
		ELSE
			//Contatora estrela
			SD_MXP_E := FALSE;
		END_IF
		LIBERA_TRIANGULO_MXP := TRUE;
	ELSE
		SD_MXP_E := FALSE;	
		LIBERA_TRIANGULO_MXP:=FALSE;
	END_IF
	
	//TEMPO PARA ENTRAR O TRIANGULO
	TMR_ESTRELA_MXP(IN:= LIBERA_TRIANGULO_MXP, PT:= T#5S);	
	LIGA_ESTRELA_MXP := TMR_ESTRELA_MXP.Q;
	//TEMPO DE INTERVALO ENTRE ESTRELA E TRIANGULO
	TMR_RETARDO_TRIANGULO_MXP(IN:= LIGA_ESTRELA_MXP, PT:= T#0.2S);
	LIGA_TRIANGULO_MXP := TMR_RETARDO_TRIANGULO_MXP.Q;
	SD_MXP_T:= LIGA_TRIANGULO_MXP;
	
	IF LIGA_MEXEDOR = TRUE THEN
		SD_MXP_P := TRUE;
	ELSE
		SD_MXP_P := FALSE;
	END_IF
		

//Fluximetro de agua ==============================================================


//gera pulso de contagem da agua		
PULSO_AGUA(CLK:=ED_FLXAGUA);

//reset contador
IF RESET_AGUA_AUTO = TRUE OR BTS_ZERAFLUXIMETRO = TRUE THEN
	RESET_AGUA := TRUE;
END_IF
//_________________________INCLUIDO________ROBY
//Calcula a quantidade de pulso para dosagem de agua, pois o preset é em litros

//Vazão da bomba 8,8L/s multiplica por 1000 pois a base de tempo é em milisegundos.
		

	QNTDADE_PULSOS_AGUA_REAL:= ((PRST_QNTDE_AGUA / 5.32 ) * 1000);
	QNTDADE_PULSOS_AGUA:= ANY_TO_TIME(QNTDADE_PULSOS_AGUA_REAL);
	
CONTADOR_AGUA(IN:= SD_BAG, PT:= QNTDADE_PULSOS_AGUA);
ET:=CONTADOR_AGUA.ET;

TMR_AGUA_DOSADA := TIME_TO_REAL(ET);
QTD_AGUA_DOSADA:= TMR_AGUA_DOSADA /1000 *  5.32;


IF SD_BAG = FALSE  THEN
	QTD_AGUA_DOSADA := PRST_QNTDE_AGUA;
END_IF

IF CNT_SEQUENCIA_SLURRY = 11 THEN
		QTD_AGUA_DOSADA := 0;
END_IF

//_________________________INCLUIDO________ROBY

//_________________________EXCLUIDO________ROBY
//Calcula a quantidade de pulso para dosagem de agua, pois o preset é em litros
//QNTDADE_PULSOS_AGUA:= REAL_TO_INT((PRST_QNTDE_AGUA / 1.67) - 3);
	
//CONTADOR_AGUA(CU:= PULSO_AGUA.Q, RESET:= RESET_AGUA,PV:=QNTDADE_PULSOS_AGUA);
//CV:=CONTADOR_AGUA.CV;
	
//QTD_AGUA_DOSADA:=cv * 1.67;
//_________________________EXCLUIDO________ROBY
	
// Manual = quando der a quantidade desejada desliga agua.
IF  CONTADOR_AGUA.Q = TRUE AND BTS_MASLU = FALSE THEN
	SD_BAG := FALSE;
END_IF

// Automatico = quando der a quantidade desejada desliga agua e incrementa o contador de posição.
IF  CONTADOR_AGUA.Q = TRUE AND BTS_MASLU = TRUE AND AGUA_DOSADA = FALSE THEN
	SD_BAG := FALSE;
	CNT_SEQUENCIA_SLURRY := CNT_SEQUENCIA_SLURRY + 1; //incrementa a sequencia
	INTERVALO_TROCA_SEQUE := TRUE; 					 // ativa retardo de inicio da sequencia, para limpar as roscas
	CONTINUA_SEQUENCIA :=FALSE;	
	AGUA_DOSADA := TRUE;
END_IF


// Automatico = segurança caso o fluximetro trave para não ficar ligada a bomba de água

//IF  BTS_MASLU = TRUE AND SD_BAG = TRUE THEN
	//TEMP_BB_AGUA(IN:= SD_BAG, PT:= T#50S);	
	//SD_BAG := TEMP_BB_AGUA.Q;

//END_IF
	
//zera volume de agua dosda
IF RESET_AGUA = TRUE THEN
	QTD_AGUA_DOSADA := 0;
	BTS_ZERAFLUXIMETRO:= FALSE;
	RESET_AGUA_AUTO := FALSE;	
	RESET_AGUA := FALSE;
	AGUA_DOSADA := FALSE;
END_IF



//Bombas materiais ===========================================================================
//Liga junto com os comandos de valvula

//Bomba de Soda
IF SD_BLL1L = TRUE OR SD_BLL1R = TRUE THEN
	SD_BSOD := TRUE;
ELSE
	SD_BSOD := FALSE;	
END_IF

//Bomba de Sulfonico
IF SD_BLL2L = TRUE OR SD_BLL2R = TRUE THEN
	SD_BSUL := TRUE;
ELSE
	SD_BSUL := FALSE;	
END_IF

//Bomba de Silicato
IF SD_BLL3L = TRUE OR SD_BLL3R = TRUE THEN
	SD_BSIL := TRUE;
ELSE
	SD_BSIL := FALSE;	
END_IF
	
//Bomba de Blend
IF SD_BLL4L = TRUE OR SD_BLL4R = TRUE THEN
	SD_BBD := TRUE;
ELSE
	SD_BBD := FALSE;	
END_IF


//===============================================================================================================
//                      Grava produção 
//===============================================================================================================

//Balança de Solido 1 
IF PRST_POSSEQ_BLS1 > 0 THEN
	//gera pulso de balansa solido 1 carregada	
	PULSO_BLS1_CARREGADA(CLK:=BLS1_CARREGADA);
	IF PULSO_BLS1_CARREGADA.Q = TRUE THEN
		LEITURA_PESO_GRAVADO_BLS1 := LEITURA_PESO_BLS1;
		LEITURA_REALIZADA_BLS1 := TRUE;
	END_IF
ELSE
	LEITURA_REALIZADA_BLS1 := TRUE;
	LEITURA_PESO_GRAVADO_BLS1 := 0;
END_IF

//Balança de Solido 2 
IF PRST_POSSEQ_BLS2 > 0 THEN
	//gera pulso de balansa solido 2 carregada	
	PULSO_BLS2_CARREGADA(CLK:=BLS2_CARREGADA);
	IF PULSO_BLS2_CARREGADA.Q = TRUE THEN
		LEITURA_PESO_GRAVADO_BLS2 := LEITURA_PESO_BLS2;
		LEITURA_REALIZADA_BLS2 := TRUE;
	END_IF
ELSE
	LEITURA_REALIZADA_BLS2 := TRUE;
	LEITURA_PESO_GRAVADO_BLS2 := 0;
END_IF

//Balança de Solido 3 
IF PRST_POSSEQ_BLS3 > 0 THEN
	//gera pulso de balansa solido 3 carregada	
	PULSO_BLS3_CARREGADA(CLK:=BLS3_CARREGADA);
	IF PULSO_BLS3_CARREGADA.Q = TRUE THEN
		LEITURA_PESO_GRAVADO_BLS3 := LEITURA_PESO_BLS3;
		LEITURA_REALIZADA_BLS3 := TRUE;
	END_IF
ELSE
	LEITURA_REALIZADA_BLS3 := TRUE;
	LEITURA_PESO_GRAVADO_BLS3 := 0;
END_IF

//Balança de Solido 4 
IF PRST_POSSEQ_BLS4 > 0 THEN
	//gera pulso de balansa solido 1 carregada	
	PULSO_BLS4_CARREGADA(CLK:=BLS4_CARREGADA);
	IF PULSO_BLS4_CARREGADA.Q = TRUE THEN
		LEITURA_PESO_GRAVADO_BLS4 := LEITURA_PESO_BLS4;
		LEITURA_REALIZADA_BLS4 := TRUE;
	END_IF
ELSE
	LEITURA_REALIZADA_BLS4 := TRUE;
	LEITURA_PESO_GRAVADO_BLS4 := 0;
END_IF

//Balança de Solido 5 
IF PRST_POSSEQ_BLS5 > 0 THEN
	//gera pulso de balansa solido 1 carregada	
	PULSO_BLS1_CARREGADA(CLK:=BLS5_CARREGADA);
	IF PULSO_BLS5_CARREGADA.Q = TRUE THEN
		LEITURA_PESO_GRAVADO_BLS5 := LEITURA_PESO_BLS5;
		LEITURA_REALIZADA_BLS5 := TRUE;
	END_IF
ELSE
	LEITURA_REALIZADA_BLS5 := TRUE;
	LEITURA_PESO_GRAVADO_BLS5 := 0;
END_IF

//Balança de Liquido 1 
IF PRST_POSSEQ_BLL1 > 0 THEN
	//gera pulso de balansa liquido 1 carregada	
	PULSO_BLL1_CARREGADA(CLK:=BLL1_CARREGADA);
	IF PULSO_BLL1_CARREGADA.Q = TRUE THEN
		LEITURA_PESO_GRAVADO_BLL1 := LEITURA_PESO_BLL1;
		LEITURA_REALIZADA_BLL1 := TRUE;
	END_IF
ELSE
	LEITURA_REALIZADA_BLL1 := TRUE;
	LEITURA_PESO_GRAVADO_BLL1 := 0;
END_IF

//Balança de Liquido 2 
IF PRST_POSSEQ_BLL2 > 0 THEN
	//gera pulso de balansa liquido 1 carregada	
	PULSO_BLL2_CARREGADA(CLK:=BLL2_CARREGADA);
	IF PULSO_BLL2_CARREGADA.Q = TRUE THEN
		LEITURA_PESO_GRAVADO_BLL2 := LEITURA_PESO_BLL2;
		LEITURA_REALIZADA_BLL2 := TRUE;
	END_IF
ELSE
	LEITURA_REALIZADA_BLL2 := TRUE;
	LEITURA_PESO_GRAVADO_BLL2 := 0;
END_IF

//Balança de Liquido 3 
IF PRST_POSSEQ_BLL3 > 0 THEN
	//gera pulso de balansa liquido 1 carregada	
	PULSO_BLL3_CARREGADA(CLK:=BLL3_CARREGADA);
	IF PULSO_BLL3_CARREGADA.Q = TRUE THEN
		LEITURA_PESO_GRAVADO_BLL3 := LEITURA_PESO_BLL3;
		LEITURA_REALIZADA_BLL3 := TRUE;		
	END_IF
ELSE
	LEITURA_REALIZADA_BLL3 := TRUE;
	LEITURA_PESO_GRAVADO_BLL3 := 0;
END_IF

//Balança de Liquido 4 
IF PRST_POSSEQ_BLL4 > 0 THEN
	//gera pulso de balansa liquido 1 carregada	
	PULSO_BLL4_CARREGADA(CLK:=BLL4_CARREGADA);
	IF PULSO_BLL4_CARREGADA.Q = TRUE THEN
		LEITURA_PESO_GRAVADO_BLL4 := LEITURA_PESO_BLL4;
		LEITURA_REALIZADA_BLL4 := TRUE;
	END_IF
ELSE
	LEITURA_REALIZADA_BLL4 := TRUE;	
	LEITURA_PESO_GRAVADO_BLL4 := 0;
END_IF

//Agua
IF CONTADOR_AGUA.Q = TRUE  THEN
	LEITURA_PESO_GRAVADO_AGUA := QTD_AGUA_DOSADA;
	LEITURA_REALIZADA_AGUA := TRUE;
END_IF


//Informa que todas as leituras foram realizadas
IF LEITURA_REALIZADA_BLS1 = TRUE AND LEITURA_REALIZADA_BLS2 = TRUE AND LEITURA_REALIZADA_BLS3 = TRUE AND LEITURA_REALIZADA_BLS4 = TRUE AND LEITURA_REALIZADA_BLS5 = TRUE
AND LEITURA_REALIZADA_BLL1 = TRUE AND LEITURA_REALIZADA_BLL2 = TRUE AND LEITURA_REALIZADA_BLL3 = TRUE AND LEITURA_REALIZADA_BLL4 = TRUE AND LEITURA_REALIZADA_AGUA = TRUE THEN
	LEITURA_STATUS_PESOS_SLURRY_GRAVADO := 1;
END_IF

//Reset status e pesos
IF PRST_RESET_STATUS_LEITURA_SLURRY = 1 THEN	
	LEITURA_REALIZADA_BLS1 := FALSE;
	LEITURA_REALIZADA_BLS2 := FALSE;
	LEITURA_REALIZADA_BLS3 := FALSE;
	LEITURA_REALIZADA_BLS4 := FALSE;
	LEITURA_REALIZADA_BLS5 := FALSE;
	LEITURA_REALIZADA_BLL1 := FALSE;
	LEITURA_REALIZADA_BLL2 := FALSE;
	LEITURA_REALIZADA_BLL3 := FALSE;
	LEITURA_REALIZADA_BLL4 := FALSE;
	LEITURA_REALIZADA_AGUA := FALSE;
	LEITURA_STATUS_PESOS_SLURRY_GRAVADO := 0;
	PRST_RESET_STATUS_LEITURA_SLURRY := 0;
END_IF

END_PROGRAM

// Device/Application/Alarmes
PROGRAM Alarmes
VAR
	//Tempos
	
	//Tempo alarme rosca de pó 1 
	TMR_TEMPO_ALARME_RPO1:TON;
	//Tempo alarme rosca de pó 2 
	TMR_TEMPO_ALARME_RPO2:TON;
	//Tempo alarme rosca de pó 3 
	TMR_TEMPO_ALARME_RPO3:TON;
	//Tempo alarme rosca de pó 4 
	TMR_TEMPO_ALARME_RPO4:TON;
	//Tempo alarme rosca de pó 5 
	TMR_TEMPO_ALARME_RPO5:TON;
	//Tempo alarme rosca 6 Horizontal 
	TMR_TEMPO_ALARME_R6:TON;
	//Tempo alarme rosca 7 Inclinada
	TMR_TEMPO_ALARME_R7:TON;
	//Tempo alarme Valvula Carga lenta BLL1
	TMR_TEMPO_ALARME_VAL_CARLENTA_BLL1:TON;
	//Tempo alarme Valvula Carga lenta BLL2
	TMR_TEMPO_ALARME_VAL_CARLENTA_BLL2:TON;
	//Tempo alarme Valvula Carga lenta BLL3
	TMR_TEMPO_ALARME_VAL_CARLENTA_BLL3:TON;
	//Tempo alarme Valvula Carga lenta BLL4
	TMR_TEMPO_ALARME_VAL_CARLENTA_BLL4:TON;
	//Tempo alarme Valvula Carga Rapida BLL1
	TMR_TEMPO_ALARME_VAL_CARRAPIDA_BLL1:TON;
	//Tempo alarme Valvula Carga Rapida BLL2
	TMR_TEMPO_ALARME_VAL_CARRAPIDA_BLL2:TON;
	//Tempo alarme Valvula Carga Rapida BLL3
	TMR_TEMPO_ALARME_VAL_CARRAPIDA_BLL3:TON;
	//Tempo alarme Valvula Carga Rapida BLL4
	TMR_TEMPO_ALARME_VAL_CARRAPIDA_BLL4:TON;
	//Tempo alarme Descarga BLS1
	TMR_TEMPO_ALARME_DESCARGA_BLS1:TON;	
	//Tempo alarme Descarga BLS2
	TMR_TEMPO_ALARME_DESCARGA_BLS2:TON;	
	//Tempo alarme Descarga BLS3
	TMR_TEMPO_ALARME_DESCARGA_BLS3:TON;	
	//Tempo alarme Descarga BLS4
	TMR_TEMPO_ALARME_DESCARGA_BLS4:TON;	
	//Tempo alarme Descarga BLS5
	TMR_TEMPO_ALARME_DESCARGA_BLS5:TON;	
	//Tempo alarme Valvula Descarga BLL1
	TMR_TEMPO_ALARME_VAL_DESCARGA_BLL1:TON;	
	//Tempo alarme Valvula Descarga BLL2
	TMR_TEMPO_ALARME_VAL_DESCARGA_BLL2:TON;
	//Tempo alarme Valvula Descarga BLL3
	TMR_TEMPO_ALARME_VAL_DESCARGA_BLL3:TON;
	//Tempo alarme Valvula Descarga BLL4
	TMR_TEMPO_ALARME_VAL_DESCARGA_BLL4:TON;
	//Tempo alarme bomba de alimentação de oleo
	TMR_TEMPO_ALARME_BOMBA_ALIM_OLEO:TON;
	//Tempo alarme Exaustor FM2 estrela
	TMR_TEMPO_ALARME_FM2_E:TON;
	//Tempo alarme Exuastor FM2 triangulo
	TMR_TEMPO_ALARME_FM2_T:TON;
	//Tempo alarme Ventilador FM2 estrela
	TMR_TEMPO_ALARME_VFM2_E:TON;
	//Tempo alarme Ventilador FM2 triangulo
	TMR_TEMPO_ALARME_VFM2_T:TON;
	//Tempo alarme esteira TC8 não entrou
	TMR_TEMPO_ALARME_ESTTC8:TON;
	//Tempo alarme peneira 1 não entrou
	TMR_TEMPO_ALARME_PN1:TON;
	//Tempo alarme peneira 2 não entrou
	TMR_TEMPO_ALARME_PN2:TON;
	//Tempo alarme peneira 3 não entrou
	TMR_TEMPO_ALARME_PN3:TON;
	//Tempo alarme peneira 4 não entrou
	TMR_TEMPO_ALARME_PN4:TON;	
	//Tempo alarme Bomba Sulfonico
	TMR_TEMPO_ALARME_BBSULFONICO:TON;
	//Tempo alarme Bomba Soda
	TMR_TEMPO_ALARME_BBSODA:TON;
	//Tempo alarme Bomba Silicato
	TMR_TEMPO_ALARME_BBSILICATO:TON;
	//Tempo alarme Bomba Agua
	TMR_TEMPO_ALARME_BBAGUA:TON;
	//Tempo alarme Bomba Blend
	TMR_TEMPO_ALARME_BBBLEND:TON;	
	//tempo alarme elevador 2 não ligou
	T_Alarme_EL2: TON;
	//tempo alarme esteira saida air lift não ligou
	T_Alarme_ESTSAIRLF: TON;
	//tempo alarme esteira saida torre não ligou
	T_Alarme_ESTSTORRE: TON;	
	//Tempo de descarga balanca solido 1
	TMR_DESCARGA_ALARME_BLS1:TON;
	//Tempo de descarga balanca solido 2
	TMR_DESCARGA_ALARME_BLS2:TON;
	//Tempo de descarga balanca solido 3
	TMR_DESCARGA_ALARME_BLS3:TON;
	//Tempo de descarga balanca solido 4
	TMR_DESCARGA_ALARME_BLS4:TON;
	//Tempo de descarga balanca solido 5
	TMR_DESCARGA_ALARME_BLS5:TON;
	//Tempo de descarga balanca liquido 1
	TMR_DESCARGA_ALARME_BLL1:TON;
	//Tempo de descarga balanca liquido 2
	TMR_DESCARGA_ALARME_BLL2:TON;
	//Tempo de descarga balanca liquido 3
	TMR_DESCARGA_ALARME_BLL3:TON;
	//Tempo de descarga balanca liquido 4
	TMR_DESCARGA_ALARME_BLL4:TON;		
	//Tempo de alarme triangulo moinho
	TMR_TRIANGULO_MOINHO_ALARME:TON;
	//Tempo de alarme estrela moinho
	TMR_ESTRELA_MOINHO_ALARME:TON;
	//Tempo de alarme esteira saida da torre	
	TMR_ESTEIRA_SAIDA_TORRE_ALARME:TON;
	//Tempo de alarme bomba de transferencia	
	TMR_BBTRANSFERENCIA_ALARME:TON;
	//Tempo de alarme falha pressao bb alta 1	
	TMR_FALHA_PRESSAO_BBALTA1_ALARME:TON;
	//Tempo de alarme falha pressao bb alta 2	
	TMR_FALHA_PRESSAO_BBALTA2_ALARME:TON;


	//Preset Tempo de alarme de descarga balanca de solido 1
	PRST_DESCARGA_BLS1_TEMP:REAL;
	//Preset Tempo de alarme de descarga balanca de solido 1
	PRST_DESCARGA_BLS1_TEMP_TIME:TIME;
	//Preset Tempo de alarme de descarga balanca de solido 2
	PRST_DESCARGA_BLS2_TEMP:REAL;
	//Preset Tempo de alarme de descarga balanca de solido 2
	PRST_DESCARGA_BLS2_TEMP_TIME:TIME;
	//Preset Tempo de alarme de descarga balanca de solido 3
	PRST_DESCARGA_BLS3_TEMP:REAL;
	//Preset Tempo de alarme de descarga balanca de solido 3
	PRST_DESCARGA_BLS3_TEMP_TIME:TIME;
	//Preset Tempo de alarme de descarga balanca de solido 4
	PRST_DESCARGA_BLS4_TEMP:REAL;
	//Preset Tempo de alarme de descarga balanca de solido 4
	PRST_DESCARGA_BLS4_TEMP_TIME:TIME;
	//Preset Tempo de alarme de descarga balanca de solido 5
	PRST_DESCARGA_BLS5_TEMP:REAL;
	//Preset Tempo de alarme de descarga balanca de solido 5
	PRST_DESCARGA_BLS5_TEMP_TIME:TIME;
	//Preset Tempo de alarme de descarga balanca de liquido 1
	PRST_DESCARGA_BLL1_TEMP:REAL;
	//Preset Tempo de alarme de descarga balanca de liquido 1
	PRST_DESCARGA_BLL1_TEMP_TIME:TIME;
	//Preset Tempo de alarme de descarga balanca de liquido 2
	PRST_DESCARGA_BLL2_TEMP:REAL;
	//Preset Tempo de alarme de descarga balanca de liquido 2
	PRST_DESCARGA_BLL2_TEMP_TIME:TIME;
	//Preset Tempo de alarme de descarga balanca de liquido 3
	PRST_DESCARGA_BLL3_TEMP:REAL;
	//Preset Tempo de alarme de descarga balanca de liquido 3
	PRST_DESCARGA_BLL3_TEMP_TIME:TIME;
	//Preset Tempo de alarme de descarga balanca de liquido 4
	PRST_DESCARGA_BLL4_TEMP:REAL;
	//Preset Tempo de alarme de descarga balanca de liquido 4
	PRST_DESCARGA_BLL4_TEMP_TIME:TIME;
	
	//Peso com margem de erro superior BLS1
	PESO_ERRO_MAX_BLS1:REAL;
	//Peso com margem de erro superior BLS2
	PESO_ERRO_MAX_BLS2:REAL;
	//Peso com margem de erro superior BLS3
	PESO_ERRO_MAX_BLS3:REAL;
	//Peso com margem de erro superior BLS4
	PESO_ERRO_MAX_BLS4:REAL;
	//Peso com margem de erro superior BLS5
	PESO_ERRO_MAX_BLS5:REAL;
	//Peso com margem de erro superior BLL1
	PESO_ERRO_MAX_BLL1:REAL;
	//Peso com margem de erro superior BLL2
	PESO_ERRO_MAX_BLL2:REAL;
	//Peso com margem de erro superior BLL3
	PESO_ERRO_MAX_BLL3:REAL;
	//Peso com margem de erro superior BLL4
	PESO_ERRO_MAX_BLL4:REAL;
	
	//Boleanos

	//Libera tempo alarme rosca de po 1
	LIBERA_TEMPO_AL_RPO1:BOOL;
	//Libera tempo alarme rosca de po 2
	LIBERA_TEMPO_AL_RPO2:BOOL;
	//Libera tempo alarme rosca de po 3
	LIBERA_TEMPO_AL_RPO3:BOOL;
	//Libera tempo alarme rosca de po 4
	LIBERA_TEMPO_AL_RPO4:BOOL;
	//Libera tempo alarme rosca de po 5
	LIBERA_TEMPO_AL_RPO5:BOOL;
	//Libera tempo alarme rosca 6
	LIBERA_TEMPO_AL_R6:BOOL;
	//Libera tempo alarme rosca 7
	LIBERA_TEMPO_AL_R7:BOOL;
	//Libera tempo alarme Carga lenta BLL1
	LIBERA_TEMPO_AL_CARLENTA_BLL1:BOOL;
	//Libera tempo alarme Carga lenta BLL2
	LIBERA_TEMPO_AL_CARLENTA_BLL2:BOOL;
	//Libera tempo alarme Carga lenta BLL3
	LIBERA_TEMPO_AL_CARLENTA_BLL3:BOOL;
	//Libera tempo alarme Carga lenta BLL4
	LIBERA_TEMPO_AL_CARLENTA_BLL4:BOOL;
	//Libera tempo alarme Carga rapida BLL1
	LIBERA_TEMPO_AL_CARRAPIDA_BLL1:BOOL;
	//Libera tempo alarme Carga rapida BLL2
	LIBERA_TEMPO_AL_CARRAPIDA_BLL2:BOOL;
	//Libera tempo alarme Carga rapida BLL3
	LIBERA_TEMPO_AL_CARRAPIDA_BLL3:BOOL;
	//Libera tempo alarme Carga rapida BLL4
	LIBERA_TEMPO_AL_CARRAPIDA_BLL4:BOOL;
	//Libera tempo alarme Descarga BLS1
	LIBERA_TEMPO_AL_DESCARGA_BLS1:BOOL;
	//Libera tempo alarme Descarga BLS2
	LIBERA_TEMPO_AL_DESCARGA_BLS2:BOOL;
	//Libera tempo alarme Descarga BLS3
	LIBERA_TEMPO_AL_DESCARGA_BLS3:BOOL;
	//Libera tempo alarme Descarga BLS4
	LIBERA_TEMPO_AL_DESCARGA_BLS4:BOOL;
	//Libera tempo alarme Descarga BLS5
	LIBERA_TEMPO_AL_DESCARGA_BLS5:BOOL;
	//Libera tempo alarme Valvula Descarga BLL1
	LIBERA_TEMPO_AL_VAL_DESCARGA_BLL1:BOOL;
	//Libera tempo alarme Valvula Descarga BLL2
	LIBERA_TEMPO_AL_VAL_DESCARGA_BLL2:BOOL;
	//Libera tempo alarme Valvula Descarga BLL3
	LIBERA_TEMPO_AL_VAL_DESCARGA_BLL3:BOOL;
	//Libera tempo alarme Valvula Descarga BLL4
	LIBERA_TEMPO_AL_VAL_DESCARGA_BLL4:BOOL;
	//Libera tempo alarme triangulo moinho
	LIBERA_TEMPO_AL_TRIAN_MOINHO:BOOL;
	//Libera tempo alarme estrela moinho
	LIBERA_TEMPO_AL_ESTRELA_MOINHO:BOOL;
	//Libera tempo alarme de alimentacao de oleo
	LIBERA_TEMPO_AL_BALIOLEO:BOOL;
	//Libera tempo alarme Exaustor FM2 estrela
	LIBERA_TEMPO_AL_FM2E:BOOL;
	//Libera tempo alarme Exaustor FM2 triangulo
	LIBERA_TEMPO_AL_FM2T:BOOL;
	//Libera tempo alarme Ventilador FM2 estrela
	LIBERA_TEMPO_AL_VFM2E:BOOL;
	//Libera tempo alarme Ventilador FM2 triangulo
	LIBERA_TEMPO_AL_VFM2T:BOOL;
	//Libera tempo alarme esteira TC8 não entrou
	LIBERA_TEMPO_AL_TC8:BOOL;
	//Libera tempo alarme peneira 1 não entrou
	LIBERA_TEMPO_AL_PN1:BOOL;
	//Libera tempo alarme peneira 2 não entrou
	LIBERA_TEMPO_AL_PN2:BOOL;
	//Libera tempo alarme peneira 3 não entrou
	LIBERA_TEMPO_AL_PN3:BOOL;
	//Libera tempo alarme peneira 4 não entrou
	LIBERA_TEMPO_AL_PN4:BOOL;
	//Libera tempo alarme elevador 2 não entrou
	LIBERA_TEMPO_AL_EL2:BOOL;
	//Libera tempo alarme esteira saida air lift não entrou
	LIBERA_TEMPO_AL_ESTSAIRLF:BOOL;
	//Libera tempo alarme esteira saida torre não entrou
	LIBERA_TEMPO_AL_ESTSTORRE:BOOL;
	//Libera tempo alarme bomba sulfonico
	LIBERA_TEMPO_AL_BBSULFONICO:BOOL;
	//Libera tempo alarme bomba soda
	LIBERA_TEMPO_AL_BBSODA:BOOL;
	//Libera tempo alarme bomba Silicato
	LIBERA_TEMPO_AL_BBSILICATO:BOOL;
	//Libera tempo alarme bomba Agua
	LIBERA_TEMPO_AL_BBAGUA:BOOL;
	//Libera tempo alarme bomba Blend
	LIBERA_TEMPO_AL_BBBLEND:BOOL;
	//Libera tempo alarme bomba transferencia
	LIBERA_TEMPO_AL_BBTRANSFE:BOOL;
	//Libera tempo alarme falha de pressao bb alta 1
	LIBERA_TEMPO_AL_FALHA_PRESSAO_BBALTA1:BOOL;
	//Libera tempo alarme falha de pressao bb alta 2
	LIBERA_TEMPO_AL_FALHA_PRESSAO_BBALTA2:BOOL;
	
	
	TEMP_AL_SIR_DOSADORES: TON;
	LIBERA_TEMP_AL_SIR_DOSADORES: BOOL;
	BLINK_ALARMES: BLINK;
	ATUALIZA_ALARMES: BOOL;
	BLINK_SIRENE: BLINK;
END_VAR

// ================================ Alarme Geral =============================================

IF  ED_BTEMER = FALSE OR ED_FTF = TRUE  THEN
	AL_GERAL := TRUE;
ELSE
	AL_GERAL := FALSE;
END_IF 

//================================= Roscas de pó ============================================

//rosca pó 1
IF SD_RPO1 = TRUE AND ED_RPO1_L = FALSE THEN
	LIBERA_TEMPO_AL_RPO1:=TRUE;
ELSE
	LIBERA_TEMPO_AL_RPO1:= FALSE;
END_IF

TMR_TEMPO_ALARME_RPO1(IN:=LIBERA_TEMPO_AL_RPO1, PT:=T#15S);

IF TMR_TEMPO_ALARME_RPO1.Q = TRUE THEN
	AL_RPO1:=TRUE;
END_IF

//rosca pó 2
IF SD_RPO2 = TRUE AND ED_RPO2_L = FALSE THEN
	LIBERA_TEMPO_AL_RPO2:=TRUE;
ELSE
	LIBERA_TEMPO_AL_RPO2:= FALSE;
END_IF

TMR_TEMPO_ALARME_RPO2(IN:=LIBERA_TEMPO_AL_RPO2, PT:=T#15S);

IF TMR_TEMPO_ALARME_RPO2.Q = TRUE THEN
	AL_RPO2:=TRUE;
END_IF

//rosca pó 3
IF SD_RPO3 = TRUE AND ED_RPO3_L = FALSE THEN
	LIBERA_TEMPO_AL_RPO3:=TRUE;
ELSE
	LIBERA_TEMPO_AL_RPO3:= FALSE;
END_IF

TMR_TEMPO_ALARME_RPO3(IN:=LIBERA_TEMPO_AL_RPO3, PT:=T#15S);

IF TMR_TEMPO_ALARME_RPO3.Q = TRUE THEN
	AL_RPO3:=TRUE;
END_IF

//rosca pó 4
IF SD_RPO4 = TRUE AND ED_RPO4_L = FALSE THEN
	LIBERA_TEMPO_AL_RPO4:=TRUE;
ELSE
	LIBERA_TEMPO_AL_RPO4:= FALSE;
END_IF

TMR_TEMPO_ALARME_RPO4(IN:=LIBERA_TEMPO_AL_RPO4, PT:=T#15S);

IF TMR_TEMPO_ALARME_RPO4.Q = TRUE THEN
	AL_RPO4:=TRUE;
END_IF

//rosca pó 5
IF SD_RPO5 = TRUE AND ED_RPO5_L = FALSE THEN
	LIBERA_TEMPO_AL_RPO5:=TRUE;
ELSE
	LIBERA_TEMPO_AL_RPO5:= FALSE;
END_IF

TMR_TEMPO_ALARME_RPO5(IN:=LIBERA_TEMPO_AL_RPO5, PT:=T#15S);

IF TMR_TEMPO_ALARME_RPO5.Q = TRUE THEN
	AL_RPO5:=TRUE;
END_IF

//============================ Roscas ========================================================

//rosca 6
IF SD_R6 = TRUE AND ED_RC6H_L = FALSE THEN
	LIBERA_TEMPO_AL_R6:=TRUE;
ELSE
	LIBERA_TEMPO_AL_R6:= FALSE;
END_IF

TMR_TEMPO_ALARME_R6(IN:=LIBERA_TEMPO_AL_R6, PT:=T#15S);

IF TMR_TEMPO_ALARME_R6.Q = TRUE THEN
	AL_RC6H:=TRUE;
END_IF

//rosca 7
IF SD_R7 = TRUE AND ED_RC7I_L = FALSE THEN
	LIBERA_TEMPO_AL_R7:=TRUE;
ELSE
	LIBERA_TEMPO_AL_R7:= FALSE;
END_IF

TMR_TEMPO_ALARME_R7(IN:=LIBERA_TEMPO_AL_R7, PT:=T#15S);

IF TMR_TEMPO_ALARME_R7.Q = TRUE THEN
	AL_RC7I:=TRUE;
END_IF

//======================== Valvulas de descargas ==========================================================

//Valvula descarga Balança de Solido 1
IF SD_BLS1 = TRUE AND ED_BLS1D_L = true THEN
	LIBERA_TEMPO_AL_DESCARGA_BLS1:=TRUE;
ELSE
	LIBERA_TEMPO_AL_DESCARGA_BLS1:= FALSE;
END_IF

TMR_TEMPO_ALARME_DESCARGA_BLS1(IN:=LIBERA_TEMPO_AL_DESCARGA_BLS1, PT:=T#15S);

IF TMR_TEMPO_ALARME_DESCARGA_BLS1.Q = TRUE THEN
	AL_BLS1D:=TRUE;
END_IF

//Valvula descarga Balança de Solido 2
IF SD_BLS2 = TRUE AND ED_BLS2D_L = TRUE THEN
	LIBERA_TEMPO_AL_DESCARGA_BLS2:=TRUE;
ELSE
	LIBERA_TEMPO_AL_DESCARGA_BLS2:= FALSE;
END_IF

TMR_TEMPO_ALARME_DESCARGA_BLS2(IN:=LIBERA_TEMPO_AL_DESCARGA_BLS2, PT:=T#15S);

IF TMR_TEMPO_ALARME_DESCARGA_BLS2.Q = TRUE THEN
	AL_BLS2D:=TRUE;
END_IF

//Valvula descarga Balança de Solido 3
IF SD_BLS3 = TRUE AND ED_BLS3D_L = TRUE THEN
	LIBERA_TEMPO_AL_DESCARGA_BLS3:=TRUE;
ELSE
	LIBERA_TEMPO_AL_DESCARGA_BLS3:= FALSE;
END_IF

TMR_TEMPO_ALARME_DESCARGA_BLS3(IN:=LIBERA_TEMPO_AL_DESCARGA_BLS3, PT:=T#15S);

IF TMR_TEMPO_ALARME_DESCARGA_BLS3.Q = TRUE THEN
	AL_BLS3D:=TRUE;
END_IF

//Valvula descarga Balança de Solido 4
IF SD_BLS4 = TRUE AND ED_BLS4D_L = TRUE THEN
	LIBERA_TEMPO_AL_DESCARGA_BLS4:=TRUE;
ELSE
	LIBERA_TEMPO_AL_DESCARGA_BLS4:= FALSE;
END_IF

TMR_TEMPO_ALARME_DESCARGA_BLS4(IN:=LIBERA_TEMPO_AL_DESCARGA_BLS4, PT:=T#15S);

IF TMR_TEMPO_ALARME_DESCARGA_BLS4.Q = TRUE THEN
	AL_BLS4D:=TRUE;
END_IF

//Valvula descarga Balança de Solido 5
IF SD_BLS5 = TRUE AND ED_BLS5D_L = TRUE THEN
	LIBERA_TEMPO_AL_DESCARGA_BLS5:=TRUE;
ELSE
	LIBERA_TEMPO_AL_DESCARGA_BLS5:= FALSE;
END_IF

TMR_TEMPO_ALARME_DESCARGA_BLS5(IN:=LIBERA_TEMPO_AL_DESCARGA_BLS5, PT:=T#15S);

IF TMR_TEMPO_ALARME_DESCARGA_BLS5.Q = TRUE THEN
	AL_BLS5D:=TRUE;
END_IF

//Valvula descarga Balança de Liquido 1
IF SD_BLL1D = TRUE AND ED_BL1D_L = FALSE THEN
	LIBERA_TEMPO_AL_VAL_DESCARGA_BLL1:=TRUE;
ELSE
	LIBERA_TEMPO_AL_VAL_DESCARGA_BLL1:= FALSE;
END_IF

TMR_TEMPO_ALARME_VAL_DESCARGA_BLL1(IN:=LIBERA_TEMPO_AL_VAL_DESCARGA_BLL1, PT:=T#15S);

IF TMR_TEMPO_ALARME_VAL_DESCARGA_BLL1.Q = TRUE THEN
	AL_BL1D:=TRUE;
END_IF

//Valvula descarga Balança de Liquido 2
IF SD_BLL2D = TRUE AND ED_BL2D_L = FALSE THEN
	LIBERA_TEMPO_AL_VAL_DESCARGA_BLL2:=TRUE;
ELSE
	LIBERA_TEMPO_AL_VAL_DESCARGA_BLL2:= FALSE;
END_IF

TMR_TEMPO_ALARME_VAL_DESCARGA_BLL2(IN:=LIBERA_TEMPO_AL_VAL_DESCARGA_BLL2, PT:=T#15S);

IF TMR_TEMPO_ALARME_VAL_DESCARGA_BLL2.Q = TRUE THEN
	AL_BL2D:=TRUE;
END_IF

//Valvula descarga Balança de Liquido 3
IF SD_BLL3D = TRUE AND ED_BL3D_L = FALSE THEN
	LIBERA_TEMPO_AL_VAL_DESCARGA_BLL3:=TRUE;
ELSE
	LIBERA_TEMPO_AL_VAL_DESCARGA_BLL3:= FALSE;
END_IF

TMR_TEMPO_ALARME_VAL_DESCARGA_BLL3(IN:=LIBERA_TEMPO_AL_VAL_DESCARGA_BLL3, PT:=T#15S);

IF TMR_TEMPO_ALARME_VAL_DESCARGA_BLL3.Q = TRUE THEN
	AL_BL3D:=TRUE;
END_IF

//Valvula descarga Balança de Liquido 4
IF SD_BLL4D = TRUE AND ED_BL4D_L = FALSE THEN
	LIBERA_TEMPO_AL_VAL_DESCARGA_BLL4:=TRUE;
ELSE
	LIBERA_TEMPO_AL_VAL_DESCARGA_BLL4:= FALSE;
END_IF

TMR_TEMPO_ALARME_VAL_DESCARGA_BLL4(IN:=LIBERA_TEMPO_AL_VAL_DESCARGA_BLL4, PT:=T#15S);

IF TMR_TEMPO_ALARME_VAL_DESCARGA_BLL4.Q = TRUE THEN
	AL_BL4D:=TRUE;
END_IF

//===================== Valvulas de carga rapida e lenta ==================================================
 
//Valvula carga Lenta Balança de Liquido 1
IF SD_BLL1L = TRUE AND ED_BLL1L_L = FALSE THEN
	LIBERA_TEMPO_AL_CARLENTA_BLL1:=TRUE;
ELSE
	LIBERA_TEMPO_AL_CARLENTA_BLL1:= FALSE;
END_IF

TMR_TEMPO_ALARME_VAL_CARLENTA_BLL1(IN:=LIBERA_TEMPO_AL_CARLENTA_BLL1, PT:=T#15S);

IF TMR_TEMPO_ALARME_VAL_CARLENTA_BLL1.Q = TRUE THEN
	AL_BLL1L:=TRUE;
END_IF

//Valvula carga Lenta Balança de Liquido 2
IF SD_BLL2L = TRUE AND ED_BLL2L_L = FALSE THEN
	LIBERA_TEMPO_AL_CARLENTA_BLL2:=TRUE;
ELSE
	LIBERA_TEMPO_AL_CARLENTA_BLL2:= FALSE;
END_IF

TMR_TEMPO_ALARME_VAL_CARLENTA_BLL2(IN:=LIBERA_TEMPO_AL_CARLENTA_BLL2, PT:=T#15S);

IF TMR_TEMPO_ALARME_VAL_CARLENTA_BLL2.Q = TRUE THEN
	AL_BLL2L:=TRUE;
END_IF

//Valvula carga Lenta Balança de Liquido 3
IF SD_BLL3L = TRUE AND ED_BLL3L_L = FALSE THEN
	LIBERA_TEMPO_AL_CARLENTA_BLL3:=TRUE;
ELSE
	LIBERA_TEMPO_AL_CARLENTA_BLL3:= FALSE;
END_IF

TMR_TEMPO_ALARME_VAL_CARLENTA_BLL3(IN:=LIBERA_TEMPO_AL_CARLENTA_BLL3, PT:=T#15S);

IF TMR_TEMPO_ALARME_VAL_CARLENTA_BLL3.Q = TRUE THEN
	AL_BLL3L:=TRUE;
END_IF

//Valvula carga Lenta Balança de Liquido 4
IF SD_BLL4L = TRUE AND ED_BLL4L_L = FALSE THEN
	LIBERA_TEMPO_AL_CARLENTA_BLL4:=TRUE;
ELSE
	LIBERA_TEMPO_AL_CARLENTA_BLL4:= FALSE;
END_IF

TMR_TEMPO_ALARME_VAL_CARLENTA_BLL4(IN:=LIBERA_TEMPO_AL_CARLENTA_BLL4, PT:=T#15S);

IF TMR_TEMPO_ALARME_VAL_CARLENTA_BLL4.Q = TRUE THEN
	AL_BLL4L:=TRUE;
END_IF

//Valvula carga Rapida Balança de Liquido 1
IF SD_BLL1R = TRUE AND ED_BLL1R_L = FALSE THEN
	LIBERA_TEMPO_AL_CARRAPIDA_BLL1:=TRUE;
ELSE
	LIBERA_TEMPO_AL_CARRAPIDA_BLL1:= FALSE;
END_IF

TMR_TEMPO_ALARME_VAL_CARRAPIDA_BLL1(IN:=LIBERA_TEMPO_AL_CARRAPIDA_BLL1, PT:=T#15S);

IF TMR_TEMPO_ALARME_VAL_CARRAPIDA_BLL1.Q = TRUE THEN
	AL_BLL1R:=TRUE;
END_IF

//Valvula carga Rapida Balança de Liquido 2
IF SD_BLL2R = TRUE AND ED_BLL2R_L = FALSE THEN
	LIBERA_TEMPO_AL_CARRAPIDA_BLL2:=TRUE;
ELSE
	LIBERA_TEMPO_AL_CARRAPIDA_BLL2:= FALSE;
END_IF

TMR_TEMPO_ALARME_VAL_CARRAPIDA_BLL2(IN:=LIBERA_TEMPO_AL_CARRAPIDA_BLL2, PT:=T#15S);

IF TMR_TEMPO_ALARME_VAL_CARRAPIDA_BLL2.Q = TRUE THEN
	AL_BLL2R:=TRUE;
END_IF

//Valvula carga Rapida Balança de Liquido 3
IF SD_BLL3R = TRUE AND ED_BLL3R_L = FALSE THEN
	LIBERA_TEMPO_AL_CARRAPIDA_BLL3:=TRUE;
ELSE
	LIBERA_TEMPO_AL_CARRAPIDA_BLL3:= FALSE;
END_IF

TMR_TEMPO_ALARME_VAL_CARRAPIDA_BLL3(IN:=LIBERA_TEMPO_AL_CARRAPIDA_BLL3, PT:=T#15S);

IF TMR_TEMPO_ALARME_VAL_CARRAPIDA_BLL3.Q = TRUE THEN
	AL_BLL3R:=TRUE;
END_IF

//Valvula carga Rapida Balança de Liquido 4
IF SD_BLL4R = TRUE AND ED_BLL4R_L = FALSE THEN
	LIBERA_TEMPO_AL_CARRAPIDA_BLL4:=TRUE;
ELSE
	LIBERA_TEMPO_AL_CARRAPIDA_BLL4:= FALSE;
END_IF

TMR_TEMPO_ALARME_VAL_CARRAPIDA_BLL4(IN:=LIBERA_TEMPO_AL_CARRAPIDA_BLL4, PT:=T#15S);

IF TMR_TEMPO_ALARME_VAL_CARRAPIDA_BLL4.Q = TRUE THEN
	AL_BLL4R:=TRUE;
END_IF

//======================== Tempo de descarga das balanças do Slurry Making ultrapassado ===================

//Descarga balança de solido 1
IF ST_CICLO_PROCESSO = TRUE AND SD_BLS1 = TRUE THEN
	
	//multiplica o preset de tempo por 1000, por ser base de tempo em milisegundos
	PRST_DESCARGA_BLS1_TEMP := PRST_TEMPO_DESCARGA_BLS1 * 1000;	
	//converte para time
	PRST_DESCARGA_BLS1_TEMP_TIME:= ANY_TO_TIME(PRST_DESCARGA_BLS1_TEMP);
	//tempo de intervalo troca de numero sequencia	
	TMR_DESCARGA_ALARME_BLS1(IN:=SD_BLS1,PT:=PRST_DESCARGA_BLS1_TEMP_TIME);
	//ativa o alarme 
	AL_DESCARGA_BLS1 := TMR_DESCARGA_ALARME_BLS1.Q;
	
END_IF

//Descarga balança de solido 2
IF ST_CICLO_PROCESSO = TRUE AND SD_BLS2 = TRUE THEN
	
	//multiplica o preset de tempo por 1000, por ser base de tempo em milisegundos
	PRST_DESCARGA_BLS2_TEMP := PRST_TEMPO_DESCARGA_BLS2 * 1000;	
	//converte para time
	PRST_DESCARGA_BLS2_TEMP_TIME:= ANY_TO_TIME(PRST_DESCARGA_BLS2_TEMP);
	//tempo de intervalo troca de numero sequencia	
	TMR_DESCARGA_ALARME_BLS2(IN:=SD_BLS2,PT:=PRST_DESCARGA_BLS2_TEMP_TIME);
	//ativa o alarme 
	AL_DESCARGA_BLS2 := TMR_DESCARGA_ALARME_BLS2.Q;
	
END_IF

//Descarga balança de solido 3
IF ST_CICLO_PROCESSO = TRUE AND SD_BLS3 = TRUE THEN
	
	//multiplica o preset de tempo por 1000, por ser base de tempo em milisegundos
	PRST_DESCARGA_BLS3_TEMP := PRST_TEMPO_DESCARGA_BLS3 * 1000;	
	//converte para time
	PRST_DESCARGA_BLS3_TEMP_TIME:= ANY_TO_TIME(PRST_DESCARGA_BLS3_TEMP);
	//tempo de intervalo troca de numero sequencia	
	TMR_DESCARGA_ALARME_BLS3(IN:=SD_BLS3,PT:=PRST_DESCARGA_BLS3_TEMP_TIME);
	//ativa o alarme 
	AL_DESCARGA_BLS3 := TMR_DESCARGA_ALARME_BLS3.Q;
	
END_IF

//Descarga balança de solido 4
IF ST_CICLO_PROCESSO = TRUE AND SD_BLS4 = TRUE THEN
	
	//multiplica o preset de tempo por 1000, por ser base de tempo em milisegundos
	PRST_DESCARGA_BLS4_TEMP := PRST_TEMPO_DESCARGA_BLS4 * 1000;	
	//converte para time
	PRST_DESCARGA_BLS4_TEMP_TIME:= ANY_TO_TIME(PRST_DESCARGA_BLS4_TEMP);
	//tempo de intervalo troca de numero sequencia	
	TMR_DESCARGA_ALARME_BLS4(IN:=SD_BLS4,PT:=PRST_DESCARGA_BLS4_TEMP_TIME);
	//ativa o alarme 
	AL_DESCARGA_BLS4 := TMR_DESCARGA_ALARME_BLS4.Q;
	
END_IF

//Descarga balança de solido 5
IF ST_CICLO_PROCESSO = TRUE AND SD_BLS5 = TRUE THEN
	
	//multiplica o preset de tempo por 1000, por ser base de tempo em milisegundos
	PRST_DESCARGA_BLS5_TEMP := PRST_TEMPO_DESCARGA_BLS5 * 1000;	
	//converte para time
	PRST_DESCARGA_BLS5_TEMP_TIME:= ANY_TO_TIME(PRST_DESCARGA_BLS5_TEMP);
	//tempo de intervalo troca de numero sequencia	
	TMR_DESCARGA_ALARME_BLS5(IN:=SD_BLS5,PT:=PRST_DESCARGA_BLS5_TEMP_TIME);
	//ativa o alarme 
	AL_DESCARGA_BLS5 := TMR_DESCARGA_ALARME_BLS5.Q;
	
END_IF

//Descarga balança de liquido 1
IF ST_CICLO_PROCESSO = TRUE AND SD_BLL1D = TRUE THEN
	
	//multiplica o preset de tempo por 1000, por ser base de tempo em milisegundos
	PRST_DESCARGA_BLL1_TEMP := PRST_TEMPO_DESCARGA_BLL1 * 1000;	
	//converte para time
	PRST_DESCARGA_BLL1_TEMP_TIME:= ANY_TO_TIME(PRST_DESCARGA_BLL1_TEMP);
	//tempo de intervalo troca de numero sequencia	
	TMR_DESCARGA_ALARME_BLL1(IN:=SD_BLL1D,PT:=PRST_DESCARGA_BLL1_TEMP_TIME);
	//ativa o alarme 
	AL_DESCARGA_BLL1 := TMR_DESCARGA_ALARME_BLL1.Q;
	
END_IF

//Descarga balança de liquido 2
IF ST_CICLO_PROCESSO = TRUE AND SD_BLL2D = TRUE THEN
	
	//multiplica o preset de tempo por 1000, por ser base de tempo em milisegundos
	PRST_DESCARGA_BLL2_TEMP := PRST_TEMPO_DESCARGA_BLL2 * 1000;	
	//converte para time
	PRST_DESCARGA_BLL2_TEMP_TIME:= ANY_TO_TIME(PRST_DESCARGA_BLL2_TEMP);
	//tempo de intervalo troca de numero sequencia	
	TMR_DESCARGA_ALARME_BLL2(IN:=SD_BLL2D,PT:=PRST_DESCARGA_BLL2_TEMP_TIME);
	//ativa o alarme 
	AL_DESCARGA_BLL2 := TMR_DESCARGA_ALARME_BLL2.Q;
	
END_IF

//Descarga balança de liquido 3
IF ST_CICLO_PROCESSO = TRUE AND SD_BLL3D = TRUE THEN
	
	//multiplica o preset de tempo por 1000, por ser base de tempo em milisegundos
	PRST_DESCARGA_BLL3_TEMP := PRST_TEMPO_DESCARGA_BLL3 * 1000;	
	//converte para time
	PRST_DESCARGA_BLL3_TEMP_TIME:= ANY_TO_TIME(PRST_DESCARGA_BLL3_TEMP);
	//tempo de intervalo troca de numero sequencia	
	TMR_DESCARGA_ALARME_BLL3(IN:=SD_BLL3D,PT:=PRST_DESCARGA_BLL3_TEMP_TIME);
	//ativa o alarme 
	AL_DESCARGA_BLL3 := TMR_DESCARGA_ALARME_BLL3.Q;
	
END_IF

//Descarga balança de liquido 4
IF ST_CICLO_PROCESSO = TRUE AND SD_BLL4D = TRUE THEN
	
	//multiplica o preset de tempo por 1000, por ser base de tempo em milisegundos
	PRST_DESCARGA_BLL4_TEMP := PRST_TEMPO_DESCARGA_BLL4 * 1000;	
	//converte para time
	PRST_DESCARGA_BLL4_TEMP_TIME:= ANY_TO_TIME(PRST_DESCARGA_BLL4_TEMP);
	//tempo de intervalo troca de numero sequencia	
	TMR_DESCARGA_ALARME_BLL4(IN:=SD_BLL4D,PT:=PRST_DESCARGA_BLL4_TEMP_TIME);
	//ativa o alarme 
	AL_DESCARGA_BLL4 := TMR_DESCARGA_ALARME_BLL4.Q;
	
END_IF

//=========================== Alarme controle de peso Slurry ================================

//Balança de sólido 1
//Calculo peso com erro superior
PESO_ERRO_MAX_BLS1 := PRST_PESO_BLS1 + (PRST_PESO_BLS1 * (PRST_PORCENTAGEM_ERRO_PESO_BLS1 / 100));
//compara a banda
IF LEITURA_PESO_BLS1 > PESO_ERRO_MAX_BLS1 AND PRST_PESO_BLS1 > 0 AND BLS1_CARREGADA = TRUE AND BTS_PERMI_DESCAR_PESO_MAX_BLS1 = FALSE THEN
	AL_PESO_ALTO_BLS1 := TRUE;
ELSIF BTS_PERMI_DESCAR_PESO_MAX_BLS1 = TRUE OR PRST_PESO_BLS1 = 0 THEN	
	AL_PESO_ALTO_BLS1 := FALSE;	
END_IF

